LIN {X 0,Y 190.572,Z 604.003,A -85,B 0,C 180,E1 -22072.137,E2 -22072.137} C_VEL
LIN {X 0,Y 192.954,Z 597.043,A -85,B 0,C 180,E1 -22074.763,E2 -22074.763} C_VEL
LIN {X 0,Y 195.805,Z 588.854,A -85,B 0,C 180,E1 -22077.234,E2 -22077.234} C_VEL
LIN {X 0,Y 199.1,Z 578.871,A -85,B 0,C 180,E1 -22079.616,E2 -22079.616} C_VEL
LIN {X 0,Y 202.385,Z 567.586,A -85,B 0,C 180,E1 -22081.683,E2 -22081.683} C_VEL
LIN {X 0,Y 205.101,Z 556.526,A -85,B 0,C 180,E1 -22083.247,E2 -22083.247} C_VEL
LIN {X 0,Y 207.556,Z 544.251,A -85,B 0,C 180,E1 -22084.553,E2 -22084.553} C_VEL
LIN {X 0,Y 209.563,Z 531.232,A -85,B 0,C 180,E1 -22085.496,E2 -22085.496} C_VEL
LIN {X 0,Y 210.767,Z 517.939,A -85,B 0,C 180,E1 -22086.116,E2 -22086.116} C_VEL
LIN {X 0,Y 212.898,Z 471.939,A -85,B 0,C 180,E1 -22087.602,E2 -22087.602} C_VEL
LIN {X 0,Y 211.816,Z 464.418,A -85,B 0,C 180,E1 -22088.143,E2 -22088.143} C_VEL
LIN {X 0,Y 206.005,Z 450.045,A -85,B 0,C 180,E1 -22090.051,E2 -22090.051} C_VEL
LIN {X 0,Y 199.852,Z 437.156,A -85,B 0,C 180,E1 -22092.148,E2 -22092.148} C_VEL
LIN {X 0,Y 192.449,Z 423.923,A -85,B 0,C 180,E1 -22094.837,E2 -22094.837} C_VEL
LIN {X 0,Y 188.849,Z 418.24,A -85,B 0,C 180,E1 -22096.231,E2 -22096.231} C_VEL
LIN {X 0,Y 186.477,Z 414.323,A -85,B 0,C 180,E1 -22097.208,E2 -22097.208} C_VEL
LIN {X 0,Y 186.222,Z 413.566,A -85,B 0,C 180,E1 -22097.52,E2 -22097.52} C_VEL
LIN {X 0,Y 185.477,Z 410.874,A -85,B 0,C 180,E1 -22099.678,E2 -22099.678} C_VEL
LIN {X 0,Y 185.507,Z 410.87,A -85,B 0,C 180,E1 -22102.711,E2 -22102.711} C_VEL
LIN {X 0,Y 185.542,Z 410.868,A -85,B 0,C 180,E1 -22107.975,E2 -22107.975} C_VEL
LIN {X 0,Y 185.581,Z 410.869,A -85,B 0,C 180,E1 -22110.577,E2 -22110.577} C_VEL
LIN {X 0,Y 185.607,Z 410.861,A -85,B 0,C 180,E1 -22115.385,E2 -22115.385} C_VEL
LIN {X 0,Y 185.712,Z 410.845,A -85,B 0,C 180,E1 -22121.101,E2 -22121.101} C_VEL
LIN {X 0,Y 185.701,Z 410.845,A -85,B 0,C 180,E1 -22124.638,E2 -22124.638} C_VEL
LIN {X 0,Y 185.889,Z 410.823,A -85,B 0,C 180,E1 -22129.418,E2 -22129.418} C_VEL
LIN {X 0,Y 185.947,Z 410.822,A -85,B 0,C 180,E1 -22133.489,E2 -22133.489} C_VEL
LIN {X 0,Y 186.208,Z 410.789,A -85,B 0,C 180,E1 -22137.837,E2 -22137.837} C_VEL
LIN {X 0,Y 186.409,Z 410.757,A -85,B 0,C 180,E1 -22140,E2 -22140} C_VEL
LIN {X 0,Y 185.932,Z 410.824,A -85,B 0,C 180,E1 -22144.336,E2 -22144.336} C_VEL
LIN {X 0,Y 186.031,Z 410.813,A -85,B 0,C 180,E1 -22148.692,E2 -22148.692} C_VEL
LIN {X 0,Y 185.767,Z 410.841,A -85,B 0,C 180,E1 -22153.12,E2 -22153.12} C_VEL
LIN {X 0,Y 185.719,Z 410.842,A -85,B 0,C 180,E1 -22157.622,E2 -22157.622} C_VEL
LIN {X 0,Y 185.617,Z 410.856,A -85,B 0,C 180,E1 -22162.249,E2 -22162.249} C_VEL
LIN {X 0,Y 185.565,Z 410.865,A -85,B 0,C 180,E1 -22167.032,E2 -22167.032} C_VEL
LIN {X 0,Y 185.58,Z 410.864,A -85,B 0,C 180,E1 -22169.493,E2 -22169.493} C_VEL
LIN {X 0,Y 185.52,Z 410.869,A -85,B 0,C 180,E1 -22174.628,E2 -22174.628} C_VEL
LIN {X 0,Y 185.545,Z 410.866,A -85,B 0,C 180,E1 -22177.304,E2 -22177.304} C_VEL
LIN {X 0,Y 185.444,Z 410.885,A -85,B 0,C 180,E1 -22182.546,E2 -22182.546} C_VEL
LIN {X 0,Y 185.514,Z 411.362,A -85,B 0,C 180,E1 -22182.682,E2 -22182.682} C_VEL
LIN {X 0,Y 186.812,Z 414.259,A -85,B 0,C 180,E1 -22183.275,E2 -22183.275} C_VEL
LIN {X 0,Y 188.891,Z 416.481,A -85,B 0,C 180,E1 -22184.064,E2 -22184.064} C_VEL
LIN {X 0,Y 190.953,Z 419.676,A -85,B 0,C 180,E1 -22184.872,E2 -22184.872} C_VEL
LIN {X 0,Y 192.354,Z 421.693,A -85,B 0,C 180,E1 -22185.396,E2 -22185.396} C_VEL
LIN {X 0,Y 197.731,Z 429.638,A -85,B 0,C 180,E1 -22187.31,E2 -22187.31} C_VEL
LIN {X 0,Y 202.517,Z 437.59,A -85,B 0,C 180,E1 -22188.923,E2 -22188.923} C_VEL
LIN {X 0,Y 209.209,Z 451.677,A -85,B 0,C 180,E1 -22191.125,E2 -22191.125} C_VEL
LIN {X 0,Y 213.457,Z 462.043,A -85,B 0,C 180,E1 -22192.478,E2 -22192.478} C_VEL
LIN {X 0,Y 210.815,Z 514.231,A -85,B 0,C 180,E1 -22194.156,E2 -22194.156} C_VEL
LIN {X 0,Y 209.398,Z 527.372,A -85,B 0,C 180,E1 -22194.892,E2 -22194.892} C_VEL
LIN {X 0,Y 207.581,Z 539.225,A -85,B 0,C 180,E1 -22195.892,E2 -22195.892} C_VEL
LIN {X 0,Y 205.096,Z 551.651,A -85,B 0,C 180,E1 -22197.337,E2 -22197.337} C_VEL
LIN {X 0,Y 202.158,Z 563.282,A -85,B 0,C 180,E1 -22199.151,E2 -22199.151} C_VEL
LIN {X 0,Y 199.144,Z 573.728,A -85,B 0,C 180,E1 -22201.26,E2 -22201.26} C_VEL
LIN {X 0,Y 195.977,Z 583.471,A -85,B 0,C 180,E1 -22203.772,E2 -22203.772} C_VEL
LIN {X 0,Y 193.167,Z 591.508,A -85,B 0,C 180,E1 -22206.409,E2 -22206.409} C_VEL
LIN {X 0,Y 190.245,Z 598.918,A -85,B 0,C 180,E1 -22209.455,E2 -22209.455} C_VEL
LIN {X 0,Y 187.895,Z 604.861,A -85,B 0,C 180,E1 -22212.589,E2 -22212.589} C_VEL
LIN {X 0,Y 186.018,Z 609.557,A -85,B 0,C 180,E1 -22215.784,E2 -22215.784} C_VEL
LIN {X 0,Y 184.684,Z 613.147,A -85,B 0,C 180,E1 -22219.032,E2 -22219.032} C_VEL
LIN {X 0,Y 184.036,Z 615,A -85,B 0,C 180,E1 -22221.214,E2 -22221.214} C_VEL
LIN {X 0,Y 183.317,Z 617.38,A -85,B 0,C 180,E1 -22225.603,E2 -22225.603} C_VEL
LIN {X 0,Y 183.183,Z 617.988,A -85,B 0,C 180,E1 -22227.802,E2 -22227.802} C_VEL
LIN {X 0,Y 183.146,Z 618.215,A -85,B 0,C 180,E1 -22230,E2 -22230} C_VEL
LIN {X 0,Y 183.183,Z 618.02,A -85,B 0,C 180,E1 -22232.199,E2 -22232.199} C_VEL
LIN {X 0,Y 183.338,Z 617.336,A -85,B 0,C 180,E1 -22234.67,E2 -22234.67} C_VEL
LIN {X 0,Y 184.039,Z 615.106,A -85,B 0,C 180,E1 -22238.787,E2 -22238.787} C_VEL
LIN {X 0,Y 185.059,Z 612.234,A -85,B 0,C 180,E1 -22242.057,E2 -22242.057} C_VEL
LIN {X 0,Y 186.553,Z 608.338,A -85,B 0,C 180,E1 -22245.291,E2 -22245.291} C_VEL
LIN {X 0,Y 188.529,Z 603.311,A -85,B 0,C 180,E1 -22248.474,E2 -22248.474} C_VEL
LIN {X 0,Y 191.104,Z 596.975,A -85,B 0,C 180,E1 -22251.578,E2 -22251.578} C_VEL
LIN {X 0,Y 194.125,Z 589.049,A -85,B 0,C 180,E1 -22254.604,E2 -22254.604} C_VEL
LIN {X 0,Y 196.876,Z 580.943,A -85,B 0,C 180,E1 -22257.084,E2 -22257.084} C_VEL
LIN {X 0,Y 199.983,Z 571.112,A -85,B 0,C 180,E1 -22259.473,E2 -22259.473} C_VEL
LIN {X 0,Y 203.16,Z 560.003,A -85,B 0,C 180,E1 -22261.549,E2 -22261.549} C_VEL
LIN {X 0,Y 205.787,Z 549.112,A -85,B 0,C 180,E1 -22263.123,E2 -22263.123} C_VEL
LIN {X 0,Y 208.141,Z 537.07,A -85,B 0,C 180,E1 -22264.443,E2 -22264.443} C_VEL
LIN {X 0,Y 209.904,Z 524.47,A -85,B 0,C 180,E1 -22265.442,E2 -22265.442} C_VEL
LIN {X 0,Y 211.125,Z 511.734,A -85,B 0,C 180,E1 -22266.071,E2 -22266.071} C_VEL
LIN {X 0,Y 213.616,Z 462.302,A -85,B 0,C 180,E1 -22267.64,E2 -22267.64} C_VEL
LIN {X 0,Y 207.998,Z 448.85,A -85,B 0,C 180,E1 -22269.437,E2 -22269.437} C_VEL
LIN {X 0,Y 201.622,Z 435.906,A -85,B 0,C 180,E1 -22271.554,E2 -22271.554} C_VEL
LIN {X 0,Y 196.195,Z 427.311,A -85,B 0,C 180,E1 -22273.405,E2 -22273.405} C_VEL
LIN {X 0,Y 193.394,Z 423.203,A -85,B 0,C 180,E1 -22274.409,E2 -22274.409} C_VEL
LIN {X 0,Y 191.057,Z 419.751,A -85,B 0,C 180,E1 -22275.284,E2 -22275.284} C_VEL
LIN {X 0,Y 188.911,Z 416.491,A -85,B 0,C 180,E1 -22276.124,E2 -22276.124} C_VEL
LIN {X 0,Y 187.893,Z 415.362,A -85,B 0,C 180,E1 -22276.511,E2 -22276.511} C_VEL
LIN {X 0,Y 186.07,Z 412.941,A -85,B 0,C 180,E1 -22277.244,E2 -22277.244} C_VEL
LIN {X 0,Y 185.467,Z 410.881,A -85,B 0,C 180,E1 -22277.614,E2 -22277.614} C_VEL
LIN {X 0,Y 185.547,Z 410.861,A -85,B 0,C 180,E1 -22282.696,E2 -22282.696} C_VEL
LIN {X 0,Y 185.549,Z 410.873,A -85,B 0,C 180,E1 -22287.976,E2 -22287.976} C_VEL
LIN {X 0,Y 185.585,Z 410.859,A -85,B 0,C 180,E1 -22290.576,E2 -22290.576} C_VEL
LIN {X 0,Y 185.609,Z 410.852,A -85,B 0,C 180,E1 -22295.385,E2 -22295.385} C_VEL
LIN {X 0,Y 185.714,Z 410.839,A -85,B 0,C 180,E1 -22301.101,E2 -22301.101} C_VEL
LIN {X 0,Y 185.733,Z 410.846,A -85,B 0,C 180,E1 -22304.64,E2 -22304.64} C_VEL
LIN {X 0,Y 185.947,Z 410.822,A -85,B 0,C 180,E1 -22309.328,E2 -22309.328} C_VEL
LIN {X 0,Y 185.97,Z 410.805,A -85,B 0,C 180,E1 -22313.49,E2 -22313.49} C_VEL
LIN {X 0,Y 186.213,Z 410.779,A -85,B 0,C 180,E1 -22317.837,E2 -22317.837} C_VEL
LIN {X 0,Y 186.411,Z 410.751,A -85,B 0,C 180,E1 -22320,E2 -22320} C_VEL
LIN {X 0,Y 185.923,Z 410.816,A -85,B 0,C 180,E1 -22324.336,E2 -22324.336} C_VEL
LIN {X 0,Y 185.985,Z 410.817,A -85,B 0,C 180,E1 -22328.694,E2 -22328.694} C_VEL
LIN {X 0,Y 185.733,Z 410.844,A -85,B 0,C 180,E1 -22333.123,E2 -22333.123} C_VEL
LIN {X 0,Y 185.694,Z 410.843,A -85,B 0,C 180,E1 -22337.624,E2 -22337.624} C_VEL
LIN {X 0,Y 185.6,Z 410.854,A -85,B 0,C 180,E1 -22342.251,E2 -22342.251} C_VEL
LIN {X 0,Y 185.564,Z 410.871,A -85,B 0,C 180,E1 -22347.032,E2 -22347.032} C_VEL
LIN {X 0,Y 185.58,Z 410.868,A -85,B 0,C 180,E1 -22349.493,E2 -22349.493} C_VEL
LIN {X 0,Y 185.501,Z 410.874,A -85,B 0,C 180,E1 -22354.632,E2 -22354.632} C_VEL
LIN {X 0,Y 185.509,Z 410.876,A -85,B 0,C 180,E1 -22357.312,E2 -22357.312} C_VEL
LIN {X 0,Y 185.469,Z 410.881,A -85,B 0,C 180,E1 -22360.324,E2 -22360.324} C_VEL
LIN {X 0,Y 186.424,Z 414.148,A -85,B 0,C 180,E1 -22362.655,E2 -22362.655} C_VEL
LIN {X 0,Y 188.884,Z 418.272,A -85,B 0,C 180,E1 -22363.678,E2 -22363.678} C_VEL
LIN {X 0,Y 190.38,Z 420.612,A -85,B 0,C 180,E1 -22364.268,E2 -22364.268} C_VEL
LIN {X 0,Y 193.811,Z 426.389,A -85,B 0,C 180,E1 -22365.588,E2 -22365.588} C_VEL
LIN {X 0,Y 198.904,Z 435.374,A -85,B 0,C 180,E1 -22367.433,E2 -22367.433} C_VEL
LIN {X 0,Y 205.402,Z 448.544,A -85,B 0,C 180,E1 -22369.662,E2 -22369.662} C_VEL
LIN {X 0,Y 211.443,Z 463.227,A -85,B 0,C 180,E1 -22371.655,E2 -22371.655} C_VEL
LIN {X 0,Y 212.289,Z 465.956,A -85,B 0,C 180,E1 -22371.95,E2 -22371.95} C_VEL
LIN {X 0,Y 213.064,Z 474.223,A -85,B 0,C 180,E1 -22372.456,E2 -22372.456} C_VEL
LIN {X 0,Y 212.426,Z 487.121,A -85,B 0,C 180,E1 -22372.861,E2 -22372.861} C_VEL
LIN {X 0,Y 211.673,Z 492.962,A -85,B 0,C 180,E1 -22372.944,E2 -22372.944} C_VEL
LIN {X 0,Y 206.194,Z 511.984,A -85,B 0,C 180,E1 -22372.597,E2 -22372.597} C_VEL
LIN {X 0,Y 205.189,Z 517.818,A -85,B 0,C 180,E1 -22372.667,E2 -22372.667} C_VEL
LIN {X 0,Y 203.891,Z 531.383,A -85,B 0,C 180,E1 -22373.311,E2 -22373.311} C_VEL
LIN {X 0,Y 202.022,Z 543.459,A -85,B 0,C 180,E1 -22374.205,E2 -22374.205} C_VEL
LIN {X 0,Y 199.632,Z 555.008,A -85,B 0,C 180,E1 -22375.411,E2 -22375.411} C_VEL
LIN {X 0,Y 196.782,Z 566.323,A -85,B 0,C 180,E1 -22376.999,E2 -22376.999} C_VEL
LIN {X 0,Y 193.351,Z 577.834,A -85,B 0,C 180,E1 -22379.107,E2 -22379.107} C_VEL
LIN {X 0,Y 190.186,Z 587.102,A -85,B 0,C 180,E1 -22381.288,E2 -22381.288} C_VEL
LIN {X 0,Y 187.081,Z 595.557,A -85,B 0,C 180,E1 -22383.806,E2 -22383.806} C_VEL
LIN {X 0,Y 184.008,Z 603.957,A -85,B 0,C 180,E1 -22387.018,E2 -22387.018} C_VEL
LIN {X 0,Y 181.358,Z 610.477,A -85,B 0,C 180,E1 -22390.179,E2 -22390.179} C_VEL
LIN {X 0,Y 178.771,Z 616.564,A -85,B 0,C 180,E1 -22394.026,E2 -22394.026} C_VEL
LIN {X 0,Y 177.403,Z 620.528,A -85,B 0,C 180,E1 -22397.414,E2 -22397.414} C_VEL
LIN {X 0,Y 176.476,Z 623.458,A -85,B 0,C 180,E1 -22400.833,E2 -22400.833} C_VEL
LIN {X 0,Y 176.139,Z 624.853,A -85,B 0,C 180,E1 -22403.125,E2 -22403.125} C_VEL
LIN {X 0,Y 175.95,Z 626.459,A -85,B 0,C 180,E1 -22407.71,E2 -22407.71} C_VEL
LIN {X 0,Y 176.021,Z 626.672,A -85,B 0,C 180,E1 -22410,E2 -22410} C_VEL
LIN {X 0,Y 175.947,Z 626.286,A -85,B 0,C 180,E1 -22413.037,E2 -22413.037} C_VEL
LIN {X 0,Y 176.14,Z 624.824,A -85,B 0,C 180,E1 -22416.874,E2 -22416.874} C_VEL
LIN {X 0,Y 176.475,Z 623.416,A -85,B 0,C 180,E1 -22419.166,E2 -22419.166} C_VEL
LIN {X 0,Y 177.401,Z 620.467,A -85,B 0,C 180,E1 -22422.585,E2 -22422.585} C_VEL
LIN {X 0,Y 178.766,Z 616.48,A -85,B 0,C 180,E1 -22425.973,E2 -22425.973} C_VEL
LIN {X 0,Y 181.351,Z 610.36,A -85,B 0,C 180,E1 -22429.821,E2 -22429.821} C_VEL
LIN {X 0,Y 183.98,Z 603.849,A -85,B 0,C 180,E1 -22432.968,E2 -22432.968} C_VEL
LIN {X 0,Y 186.513,Z 596.873,A -85,B 0,C 180,E1 -22435.679,E2 -22435.679} C_VEL
LIN {X 0,Y 189.491,Z 588.683,A -85,B 0,C 180,E1 -22438.221,E2 -22438.221} C_VEL
LIN {X 0,Y 192.938,Z 578.7,A -85,B 0,C 180,E1 -22440.661,E2 -22440.661} C_VEL
LIN {X 0,Y 196.374,Z 567.414,A -85,B 0,C 180,E1 -22442.772,E2 -22442.772} C_VEL
LIN {X 0,Y 199.204,Z 556.353,A -85,B 0,C 180,E1 -22444.367,E2 -22444.367} C_VEL
LIN {X 0,Y 201.749,Z 544.077,A -85,B 0,C 180,E1 -22445.696,E2 -22445.696} C_VEL
LIN {X 0,Y 203.778,Z 531.507,A -85,B 0,C 180,E1 -22446.627,E2 -22446.627} C_VEL
LIN {X 0,Y 205.04,Z 518.252,A -85,B 0,C 180,E1 -22447.267,E2 -22447.267} C_VEL
LIN {X 0,Y 207.279,Z 472.993,A -85,B 0,C 180,E1 -22448.754,E2 -22448.754} C_VEL
LIN {X 0,Y 206.377,Z 466.975,A -85,B 0,C 180,E1 -22449.218,E2 -22449.218} C_VEL
LIN {X 0,Y 200.979,Z 453.477,A -85,B 0,C 180,E1 -22451.099,E2 -22451.099} C_VEL
LIN {X 0,Y 195.129,Z 441.074,A -85,B 0,C 180,E1 -22453.213,E2 -22453.213} C_VEL
LIN {X 0,Y 188.378,Z 428.76,A -85,B 0,C 180,E1 -22455.815,E2 -22455.815} C_VEL
LIN {X 0,Y 181.983,Z 418.515,A -85,B 0,C 180,E1 -22458.505,E2 -22458.505} C_VEL
LIN {X 0,Y 179.496,Z 414.781,A -85,B 0,C 180,E1 -22459.629,E2 -22459.629} C_VEL
LIN {X 0,Y 178.901,Z 413.578,A -85,B 0,C 180,E1 -22459.963,E2 -22459.963} C_VEL
LIN {X 0,Y 178.402,Z 411.755,A -85,B 0,C 180,E1 -22461.549,E2 -22461.549} C_VEL
LIN {X 0,Y 178.486,Z 411.749,A -85,B 0,C 180,E1 -22466.547,E2 -22466.547} C_VEL
LIN {X 0,Y 178.522,Z 411.746,A -85,B 0,C 180,E1 -22470.007,E2 -22470.007} C_VEL
LIN {X 0,Y 178.535,Z 411.745,A -85,B 0,C 180,E1 -22474.876,E2 -22474.876} C_VEL
LIN {X 0,Y 178.655,Z 411.723,A -85,B 0,C 180,E1 -22480.755,E2 -22480.755} C_VEL
LIN {X 0,Y 178.661,Z 411.723,A -85,B 0,C 180,E1 -22486.348,E2 -22486.348} C_VEL
LIN {X 0,Y 178.911,Z 411.69,A -85,B 0,C 180,E1 -22490.96,E2 -22490.96} C_VEL
LIN {X 0,Y 179.153,Z 411.668,A -85,B 0,C 180,E1 -22497.752,E2 -22497.752} C_VEL
LIN {X 0,Y 179.372,Z 411.633,A -85,B 0,C 180,E1 -22500,E2 -22500} C_VEL
LIN {X 0,Y 178.88,Z 411.701,A -85,B 0,C 180,E1 -22504.507,E2 -22504.507} C_VEL
LIN {X 0,Y 178.98,Z 411.69,A -85,B 0,C 180,E1 -22509.037,E2 -22509.037} C_VEL
LIN {X 0,Y 178.69,Z 411.724,A -85,B 0,C 180,E1 -22513.65,E2 -22513.65} C_VEL
LIN {X 0,Y 178.681,Z 411.723,A -85,B 0,C 180,E1 -22518.341,E2 -22518.341} C_VEL
LIN {X 0,Y 178.532,Z 411.744,A -85,B 0,C 180,E1 -22523.182,E2 -22523.182} C_VEL
LIN {X 0,Y 178.489,Z 411.753,A -85,B 0,C 180,E1 -22528.197,E2 -22528.197} C_VEL
LIN {X 0,Y 178.48,Z 411.746,A -85,B 0,C 180,E1 -22530.791,E2 -22530.791} C_VEL
LIN {X 0,Y 178.497,Z 411.743,A -85,B 0,C 180,E1 -22534.225,E2 -22534.225} C_VEL
LIN {X 0,Y 178.431,Z 411.757,A -85,B 0,C 180,E1 -22539.796,E2 -22539.796} C_VEL
LIN {X 0,Y 178.446,Z 411.752,A -85,B 0,C 180,E1 -22540.16,E2 -22540.16} C_VEL
LIN {X 0,Y 179.377,Z 414.488,A -85,B 0,C 180,E1 -22540.685,E2 -22540.685} C_VEL
LIN {X 0,Y 181.412,Z 416.708,A -85,B 0,C 180,E1 -22541.563,E2 -22541.563} C_VEL
LIN {X 0,Y 184.264,Z 420.892,A -85,B 0,C 180,E1 -22542.796,E2 -22542.796} C_VEL
LIN {X 0,Y 185.603,Z 422.698,A -85,B 0,C 180,E1 -22543.344,E2 -22543.344} C_VEL
LIN {X 0,Y 191.446,Z 431.245,A -85,B 0,C 180,E1 -22545.62,E2 -22545.62} C_VEL
LIN {X 0,Y 197.09,Z 440.277,A -85,B 0,C 180,E1 -22547.654,E2 -22547.654} C_VEL
LIN {X 0,Y 203.052,Z 452.692,A -85,B 0,C 180,E1 -22549.747,E2 -22549.747} C_VEL
LIN {X 0,Y 207.787,Z 464.054,A -85,B 0,C 180,E1 -22551.346,E2 -22551.346} C_VEL
LIN {X 0,Y 205.089,Z 514.652,A -85,B 0,C 180,E1 -22553.007,E2 -22553.007} C_VEL
LIN {X 0,Y 203.546,Z 528.236,A -85,B 0,C 180,E1 -22553.795,E2 -22553.795} C_VEL
LIN {X 0,Y 201.56,Z 540.528,A -85,B 0,C 180,E1 -22554.878,E2 -22554.878} C_VEL
LIN {X 0,Y 199.163,Z 551.823,A -85,B 0,C 180,E1 -22556.236,E2 -22556.236} C_VEL
LIN {X 0,Y 196.107,Z 563.453,A -85,B 0,C 180,E1 -22558.089,E2 -22558.089} C_VEL
LIN {X 0,Y 192.944,Z 573.898,A -85,B 0,C 180,E1 -22560.245,E2 -22560.245} C_VEL
LIN {X 0,Y 189.715,Z 583.429,A -85,B 0,C 180,E1 -22562.759,E2 -22562.759} C_VEL
LIN {X 0,Y 186.677,Z 591.678,A -85,B 0,C 180,E1 -22565.536,E2 -22565.536} C_VEL
LIN {X 0,Y 183.624,Z 599.087,A -85,B 0,C 180,E1 -22568.679,E2 -22568.679} C_VEL
LIN {X 0,Y 181.112,Z 605.03,A -85,B 0,C 180,E1 -22571.915,E2 -22571.915} C_VEL
LIN {X 0,Y 179.134,Z 609.725,A -85,B 0,C 180,E1 -22575.226,E2 -22575.226} C_VEL
LIN {X 0,Y 177.702,Z 613.315,A -85,B 0,C 180,E1 -22578.595,E2 -22578.595} C_VEL
LIN {X 0,Y 177.033,Z 615.167,A -85,B 0,C 180,E1 -22580.863,E2 -22580.863} C_VEL
LIN {X 0,Y 176.262,Z 617.547,A -85,B 0,C 180,E1 -22585.427,E2 -22585.427} C_VEL
LIN {X 0,Y 176.099,Z 618.155,A -85,B 0,C 180,E1 -22587.713,E2 -22587.713} C_VEL
LIN {X 0,Y 176.057,Z 618.382,A -85,B 0,C 180,E1 -22590,E2 -22590} C_VEL
LIN {X 0,Y 176.099,Z 618.187,A -85,B 0,C 180,E1 -22592.288,E2 -22592.288} C_VEL
LIN {X 0,Y 176.232,Z 617.6,A -85,B 0,C 180,E1 -22594.575,E2 -22594.575} C_VEL
LIN {X 0,Y 177.036,Z 615.272,A -85,B 0,C 180,E1 -22599.137,E2 -22599.137} C_VEL
LIN {X 0,Y 178.123,Z 612.4,A -85,B 0,C 180,E1 -22602.534,E2 -22602.534} C_VEL
LIN {X 0,Y 179.703,Z 608.504,A -85,B 0,C 180,E1 -22605.889,E2 -22605.889} C_VEL
LIN {X 0,Y 181.808,Z 603.476,A -85,B 0,C 180,E1 -22609.183,E2 -22609.183} C_VEL
LIN {X 0,Y 184.519,Z 597.14,A -85,B 0,C 180,E1 -22612.389,E2 -22612.389} C_VEL
LIN {X 0,Y 187.661,Z 589.215,A -85,B 0,C 180,E1 -22615.511,E2 -22615.511} C_VEL
LIN {X 0,Y 190.501,Z 581.314,A -85,B 0,C 180,E1 -22617.999,E2 -22617.999} C_VEL
LIN {X 0,Y 193.836,Z 571.276,A -85,B 0,C 180,E1 -22620.505,E2 -22620.505} C_VEL
LIN {X 0,Y 197.151,Z 560.165,A -85,B 0,C 180,E1 -22622.628,E2 -22622.628} C_VEL
LIN {X 0,Y 199.882,Z 549.273,A -85,B 0,C 180,E1 -22624.234,E2 -22624.234} C_VEL
LIN {X 0,Y 202.318,Z 537.23,A -85,B 0,C 180,E1 -22625.582,E2 -22625.582} C_VEL
LIN {X 0,Y 204.211,Z 524.37,A -85,B 0,C 180,E1 -22626.609,E2 -22626.609} C_VEL
LIN {X 0,Y 205.488,Z 511.156,A -85,B 0,C 180,E1 -22627.262,E2 -22627.262} C_VEL
LIN {X 0,Y 207.921,Z 464.197,A -85,B 0,C 180,E1 -22628.784,E2 -22628.784} C_VEL
LIN {X 0,Y 202.209,Z 450.62,A -85,B 0,C 180,E1 -22630.725,E2 -22630.725} C_VEL
LIN {X 0,Y 196.625,Z 439.377,A -85,B 0,C 180,E1 -22632.695,E2 -22632.695} C_VEL
LIN {X 0,Y 190.415,Z 429.547,A -85,B 0,C 180,E1 -22634.965,E2 -22634.965} C_VEL
LIN {X 0,Y 184.567,Z 421.113,A -85,B 0,C 180,E1 -22637.291,E2 -22637.291} C_VEL
LIN {X 0,Y 182.337,Z 418.107,A -85,B 0,C 180,E1 -22638.234,E2 -22638.234} C_VEL
LIN {X 0,Y 181.448,Z 416.707,A -85,B 0,C 180,E1 -22638.633,E2 -22638.633} C_VEL
LIN {X 0,Y 179.397,Z 414.447,A -85,B 0,C 180,E1 -22639.523,E2 -22639.523} C_VEL
LIN {X 0,Y 178.46,Z 411.725,A -85,B 0,C 180,E1 -22640.12,E2 -22640.12} C_VEL
LIN {X 0,Y 178.499,Z 411.742,A -85,B 0,C 180,E1 -22645.775,E2 -22645.775} C_VEL
LIN {X 0,Y 178.526,Z 411.738,A -85,B 0,C 180,E1 -22650.006,E2 -22650.006} C_VEL
LIN {X 0,Y 178.538,Z 411.733,A -85,B 0,C 180,E1 -22654.876,E2 -22654.876} C_VEL
LIN {X 0,Y 178.658,Z 411.717,A -85,B 0,C 180,E1 -22660.755,E2 -22660.755} C_VEL
LIN {X 0,Y 178.68,Z 411.727,A -85,B 0,C 180,E1 -22664.018,E2 -22664.018} C_VEL
LIN {X 0,Y 178.899,Z 411.7,A -85,B 0,C 180,E1 -22669.153,E2 -22669.153} C_VEL
LIN {X 0,Y 178.935,Z 411.68,A -85,B 0,C 180,E1 -22673.233,E2 -22673.233} C_VEL
LIN {X 0,Y 179.159,Z 411.658,A -85,B 0,C 180,E1 -22677.752,E2 -22677.752} C_VEL
LIN {X 0,Y 179.374,Z 411.627,A -85,B 0,C 180,E1 -22680,E2 -22680} C_VEL
LIN {X 0,Y 178.871,Z 411.692,A -85,B 0,C 180,E1 -22684.507,E2 -22684.507} C_VEL
LIN {X 0,Y 178.914,Z 411.699,A -85,B 0,C 180,E1 -22689.04,E2 -22689.04} C_VEL
LIN {X 0,Y 178.662,Z 411.727,A -85,B 0,C 180,E1 -22693.652,E2 -22693.652} C_VEL
LIN {X 0,Y 178.627,Z 411.733,A -85,B 0,C 180,E1 -22699.216,E2 -22699.216} C_VEL
LIN {X 0,Y 178.537,Z 411.746,A -85,B 0,C 180,E1 -22705.124,E2 -22705.124} C_VEL
LIN {X 0,Y 178.48,Z 411.75,A -85,B 0,C 180,E1 -22710.791,E2 -22710.791} C_VEL
LIN {X 0,Y 178.487,Z 411.749,A -85,B 0,C 180,E1 -22714.219,E2 -22714.219} C_VEL
LIN {X 0,Y 178.411,Z 411.802,A -85,B 0,C 180,E1 -22718.449,E2 -22718.449} C_VEL
LIN {X 0,Y 179.015,Z 413.784,A -85,B 0,C 180,E1 -22720.006,E2 -22720.006} C_VEL
LIN {X 0,Y 181.346,Z 417.754,A -85,B 0,C 180,E1 -22721.106,E2 -22721.106} C_VEL
LIN {X 0,Y 182.923,Z 419.849,A -85,B 0,C 180,E1 -22721.787,E2 -22721.787} C_VEL
LIN {X 0,Y 186.834,Z 426.344,A -85,B 0,C 180,E1 -22723.461,E2 -22723.461} C_VEL
LIN {X 0,Y 191.428,Z 434.096,A -85,B 0,C 180,E1 -22725.287,E2 -22725.287} C_VEL
LIN {X 0,Y 197.531,Z 445.859,A -85,B 0,C 180,E1 -22727.575,E2 -22727.575} C_VEL
LIN {X 0,Y 203.228,Z 458.646,A -85,B 0,C 180,E1 -22729.602,E2 -22729.602} C_VEL
LIN {X 0,Y 206.798,Z 467.957,A -85,B 0,C 180,E1 -22730.843,E2 -22730.843} C_VEL
LIN {X 0,Y 207.45,Z 473.974,A -85,B 0,C 180,E1 -22731.25,E2 -22731.25} C_VEL
LIN {X 0,Y 205.189,Z 517.818,A -85,B 0,C 180,E1 -22732.667,E2 -22732.667} C_VEL
LIN {X 0,Y 204.063,Z 523.622,A -85,B 0,C 180,E1 -22732.753,E2 -22732.753} C_VEL
LIN {X 0,Y 200.646,Z 532.949,A -85,B 0,C 180,E1 -22732.763,E2 -22732.763} C_VEL
LIN {X 0,Y 196.974,Z 542.149,A -85,B 0,C 180,E1 -22732.994,E2 -22732.994} C_VEL
LIN {X 0,Y 195.437,Z 547.622,A -85,B 0,C 180,E1 -22733.41,E2 -22733.41} C_VEL
LIN {X 0,Y 192.494,Z 560.045,A -85,B 0,C 180,E1 -22734.897,E2 -22734.897} C_VEL
LIN {X 0,Y 189.231,Z 571.6,A -85,B 0,C 180,E1 -22736.782,E2 -22736.782} C_VEL
LIN {X 0,Y 185.761,Z 582.006,A -85,B 0,C 180,E1 -22738.97,E2 -22738.97} C_VEL
LIN {X 0,Y 182.607,Z 590.515,A -85,B 0,C 180,E1 -22741.243,E2 -22741.243} C_VEL
LIN {X 0,Y 179.548,Z 598.369,A -85,B 0,C 180,E1 -22743.873,E2 -22743.873} C_VEL
LIN {X 0,Y 176.493,Z 606.043,A -85,B 0,C 180,E1 -22747.154,E2 -22747.154} C_VEL
LIN {X 0,Y 173.4,Z 613.122,A -85,B 0,C 180,E1 -22751.08,E2 -22751.08} C_VEL
LIN {X 0,Y 171.36,Z 617.831,A -85,B 0,C 180,E1 -22754.538,E2 -22754.538} C_VEL
LIN {X 0,Y 170.063,Z 621.434,A -85,B 0,C 180,E1 -22758.075,E2 -22758.075} C_VEL
LIN {X 0,Y 169.435,Z 623.291,A -85,B 0,C 180,E1 -22760.449,E2 -22760.449} C_VEL
LIN {X 0,Y 169.074,Z 624.686,A -85,B 0,C 180,E1 -22762.836,E2 -22762.836} C_VEL
LIN {X 0,Y 168.859,Z 626.292,A -85,B 0,C 180,E1 -22767.614,E2 -22767.614} C_VEL
LIN {X 0,Y 168.934,Z 626.505,A -85,B 0,C 180,E1 -22770,E2 -22770} C_VEL
LIN {X 0,Y 168.85,Z 626.229,A -85,B 0,C 180,E1 -22772.627,E2 -22772.627} C_VEL
LIN {X 0,Y 169.075,Z 624.656,A -85,B 0,C 180,E1 -22777.163,E2 -22777.163} C_VEL
LIN {X 0,Y 169.434,Z 623.247,A -85,B 0,C 180,E1 -22779.55,E2 -22779.55} C_VEL
LIN {X 0,Y 170.445,Z 620.299,A -85,B 0,C 180,E1 -22783.107,E2 -22783.107} C_VEL
LIN {X 0,Y 171.925,Z 616.311,A -85,B 0,C 180,E1 -22786.627,E2 -22786.627} C_VEL
LIN {X 0,Y 174.661,Z 610.191,A -85,B 0,C 180,E1 -22790.614,E2 -22790.614} C_VEL
LIN {X 0,Y 177.551,Z 603.404,A -85,B 0,C 180,E1 -22793.988,E2 -22793.988} C_VEL
LIN {X 0,Y 180.696,Z 595.212,A -85,B 0,C 180,E1 -22797.194,E2 -22797.194} C_VEL
LIN {X 0,Y 183.95,Z 586.709,A -85,B 0,C 180,E1 -22799.78,E2 -22799.78} C_VEL
LIN {X 0,Y 187.635,Z 576.207,A -85,B 0,C 180,E1 -22802.259,E2 -22802.259} C_VEL
LIN {X 0,Y 191.286,Z 564.385,A -85,B 0,C 180,E1 -22804.394,E2 -22804.394} C_VEL
LIN {X 0,Y 194.249,Z 552.463,A -85,B 0,C 180,E1 -22806.01,E2 -22806.01} C_VEL
LIN {X 0,Y 196.749,Z 540.053,A -85,B 0,C 180,E1 -22807.23,E2 -22807.23} C_VEL
LIN {X 0,Y 198.669,Z 527.329,A -85,B 0,C 180,E1 -22808.08,E2 -22808.08} C_VEL
LIN {X 0,Y 199.785,Z 512.619,A -85,B 0,C 180,E1 -22808.683,E2 -22808.683} C_VEL
LIN {X 0,Y 201.745,Z 474.092,A -85,B 0,C 180,E1 -22809.969,E2 -22809.969} C_VEL
LIN {X 0,Y 201.098,Z 469.719,A -85,B 0,C 180,E1 -22810.322,E2 -22810.322} C_VEL
LIN {X 0,Y 195.588,Z 455.883,A -85,B 0,C 180,E1 -22812.365,E2 -22812.365} C_VEL
LIN {X 0,Y 190.431,Z 444.902,A -85,B 0,C 180,E1 -22814.35,E2 -22814.35} C_VEL
LIN {X 0,Y 184.192,Z 433.392,A -85,B 0,C 180,E1 -22816.904,E2 -22816.904} C_VEL
LIN {X 0,Y 178.345,Z 423.803,A -85,B 0,C 180,E1 -22819.514,E2 -22819.514} C_VEL
LIN {X 0,Y 175.055,Z 418.775,A -85,B 0,C 180,E1 -22821.103,E2 -22821.103} C_VEL
LIN {X 0,Y 171.975,Z 414.725,A -85,B 0,C 180,E1 -22822.655,E2 -22822.655} C_VEL
LIN {X 0,Y 171.494,Z 413.324,A -85,B 0,C 180,E1 -22822.993,E2 -22822.993} C_VEL
LIN {X 0,Y 171.388,Z 412.634,A -85,B 0,C 180,E1 -22823.699,E2 -22823.699} C_VEL
LIN {X 0,Y 171.44,Z 412.624,A -85,B 0,C 180,E1 -22829.414,E2 -22829.414} C_VEL
LIN {X 0,Y 171.47,Z 412.627,A -85,B 0,C 180,E1 -22834.384,E2 -22834.384} C_VEL
LIN {X 0,Y 171.611,Z 412.6,A -85,B 0,C 180,E1 -22840.875,E2 -22840.875} C_VEL
LIN {X 0,Y 171.581,Z 412.602,A -85,B 0,C 180,E1 -22845.773,E2 -22845.773} C_VEL
LIN {X 0,Y 171.848,Z 412.568,A -85,B 0,C 180,E1 -22850.585,E2 -22850.585} C_VEL
LIN {X 0,Y 171.815,Z 412.571,A -85,B 0,C 180,E1 -22855.308,E2 -22855.308} C_VEL
LIN {X 0,Y 172.334,Z 412.509,A -85,B 0,C 180,E1 -22860,E2 -22860} C_VEL
LIN {X 0,Y 171.829,Z 412.579,A -85,B 0,C 180,E1 -22864.692,E2 -22864.692} C_VEL
LIN {X 0,Y 171.912,Z 412.571,A -85,B 0,C 180,E1 -22869.412,E2 -22869.412} C_VEL
LIN {X 0,Y 171.615,Z 412.609,A -85,B 0,C 180,E1 -22874.224,E2 -22874.224} C_VEL
LIN {X 0,Y 171.576,Z 412.614,A -85,B 0,C 180,E1 -22879.591,E2 -22879.591} C_VEL
LIN {X 0,Y 171.47,Z 412.619,A -85,B 0,C 180,E1 -22885.617,E2 -22885.617} C_VEL
LIN {X 0,Y 171.443,Z 412.622,A -85,B 0,C 180,E1 -22890.587,E2 -22890.587} C_VEL
LIN {X 0,Y 171.405,Z 412.631,A -85,B 0,C 180,E1 -22896.48,E2 -22896.48} C_VEL
LIN {X 0,Y 171.395,Z 412.628,A -85,B 0,C 180,E1 -22897.308,E2 -22897.308} C_VEL
LIN {X 0,Y 172.287,Z 415.241,A -85,B 0,C 180,E1 -22897.891,E2 -22897.891} C_VEL
LIN {X 0,Y 174.273,Z 417.501,A -85,B 0,C 180,E1 -22898.874,E2 -22898.874} C_VEL
LIN {X 0,Y 175.154,Z 418.382,A -85,B 0,C 180,E1 -22899.288,E2 -22899.288} C_VEL
LIN {X 0,Y 177.141,Z 421.538,A -85,B 0,C 180,E1 -22900.268,E2 -22900.268} C_VEL
LIN {X 0,Y 178.634,Z 423.32,A -85,B 0,C 180,E1 -22900.941,E2 -22900.941} C_VEL
LIN {X 0,Y 184.738,Z 432.117,A -85,B 0,C 180,E1 -22903.582,E2 -22903.582} C_VEL
LIN {X 0,Y 191.104,Z 441.981,A -85,B 0,C 180,E1 -22906.073,E2 -22906.073} C_VEL
LIN {X 0,Y 195.197,Z 449.766,A -85,B 0,C 180,E1 -22907.608,E2 -22907.608} C_VEL
LIN {X 0,Y 200.959,Z 463.056,A -85,B 0,C 180,E1 -22909.715,E2 -22909.715} C_VEL
LIN {X 0,Y 202.19,Z 466.041,A -85,B 0,C 180,E1 -22910.148,E2 -22910.148} C_VEL
LIN {X 0,Y 199.465,Z 515.085,A -85,B 0,C 180,E1 -22911.798,E2 -22911.798} C_VEL
LIN {X 0,Y 197.842,Z 528.541,A -85,B 0,C 180,E1 -22912.589,E2 -22912.589} C_VEL
LIN {X 0,Y 195.802,Z 540.702,A -85,B 0,C 180,E1 -22913.684,E2 -22913.684} C_VEL
LIN {X 0,Y 193.313,Z 551.995,A -85,B 0,C 180,E1 -22915.069,E2 -22915.069} C_VEL
LIN {X 0,Y 190.113,Z 563.625,A -85,B 0,C 180,E1 -22916.957,E2 -22916.957} C_VEL
LIN {X 0,Y 186.817,Z 574.069,A -85,B 0,C 180,E1 -22919.165,E2 -22919.165} C_VEL
LIN {X 0,Y 183.785,Z 582.606,A -85,B 0,C 180,E1 -22921.446,E2 -22921.446} C_VEL
LIN {X 0,Y 180.853,Z 590.462,A -85,B 0,C 180,E1 -22924.076,E2 -22924.076} C_VEL
LIN {X 0,Y 177.54,Z 598.144,A -85,B 0,C 180,E1 -22927.297,E2 -22927.297} C_VEL
LIN {X 0,Y 174.356,Z 605.2,A -85,B 0,C 180,E1 -22931.188,E2 -22931.188} C_VEL
LIN {X 0,Y 172.275,Z 609.894,A -85,B 0,C 180,E1 -22934.623,E2 -22934.623} C_VEL
LIN {X 0,Y 170.746,Z 613.483,A -85,B 0,C 180,E1 -22938.124,E2 -22938.124} C_VEL
LIN {X 0,Y 170.01,Z 615.336,A -85,B 0,C 180,E1 -22940.483,E2 -22940.483} C_VEL
LIN {X 0,Y 169.18,Z 617.715,A -85,B 0,C 180,E1 -22945.235,E2 -22945.235} C_VEL
LIN {X 0,Y 169.003,Z 618.322,A -85,B 0,C 180,E1 -22947.617,E2 -22947.617} C_VEL
LIN {X 0,Y 168.971,Z 618.549,A -85,B 0,C 180,E1 -22950,E2 -22950} C_VEL
LIN {X 0,Y 169.134,Z 617.945,A -85,B 0,C 180,E1 -22954.23,E2 -22954.23} C_VEL
LIN {X 0,Y 169.455,Z 616.799,A -85,B 0,C 180,E1 -22957.148,E2 -22957.148} C_VEL
LIN {X 0,Y 170.013,Z 615.439,A -85,B 0,C 180,E1 -22959.518,E2 -22959.518} C_VEL
LIN {X 0,Y 171.18,Z 612.567,A -85,B 0,C 180,E1 -22963.051,E2 -22963.051} C_VEL
LIN {X 0,Y 172.882,Z 608.67,A -85,B 0,C 180,E1 -22966.533,E2 -22966.533} C_VEL
LIN {X 0,Y 175.121,Z 603.642,A -85,B 0,C 180,E1 -22969.946,E2 -22969.946} C_VEL
LIN {X 0,Y 177.979,Z 597.305,A -85,B 0,C 180,E1 -22973.259,E2 -22973.259} C_VEL
LIN {X 0,Y 181.176,Z 589.59,A -85,B 0,C 180,E1 -22976.406,E2 -22976.406} C_VEL
LIN {X 0,Y 184.254,Z 581.478,A -85,B 0,C 180,E1 -22979.037,E2 -22979.037} C_VEL
LIN {X 0,Y 187.742,Z 571.44,A -85,B 0,C 180,E1 -22981.607,E2 -22981.607} C_VEL
LIN {X 0,Y 191.219,Z 560.327,A -85,B 0,C 180,E1 -22983.773,E2 -22983.773} C_VEL
LIN {X 0,Y 194.068,Z 549.434,A -85,B 0,C 180,E1 -22985.411,E2 -22985.411} C_VEL
LIN {X 0,Y 196.589,Z 537.39,A -85,B 0,C 180,E1 -22986.785,E2 -22986.785} C_VEL
LIN {X 0,Y 198.6,Z 524.333,A -85,B 0,C 180,E1 -22987.838,E2 -22987.838} C_VEL
LIN {X 0,Y 199.904,Z 511.235,A -85,B 0,C 180,E1 -22988.493,E2 -22988.493} C_VEL
LIN {X 0,Y 202.35,Z 466.21,A -85,B 0,C 180,E1 -22989.978,E2 -22989.978} C_VEL
LIN {X 0,Y 196.375,Z 452.153,A -85,B 0,C 180,E1 -22992.141,E2 -22992.141} C_VEL
LIN {X 0,Y 192.033,Z 443.516,A -85,B 0,C 180,E1 -22993.768,E2 -22993.768} C_VEL
LIN {X 0,Y 186.274,Z 434.333,A -85,B 0,C 180,E1 -22995.997,E2 -22995.997} C_VEL
LIN {X 0,Y 180.714,Z 426.272,A -85,B 0,C 180,E1 -22998.334,E2 -22998.334} C_VEL
LIN {X 0,Y 177.851,Z 422.234,A -85,B 0,C 180,E1 -22999.634,E2 -22999.634} C_VEL
LIN {X 0,Y 175.528,Z 419.078,A -85,B 0,C 180,E1 -23000.739,E2 -23000.739} C_VEL
LIN {X 0,Y 174.791,Z 417.806,A -85,B 0,C 180,E1 -23001.118,E2 -23001.118} C_VEL
LIN {X 0,Y 172.684,Z 415.846,A -85,B 0,C 180,E1 -23002.129,E2 -23002.129} C_VEL
LIN {X 0,Y 171.512,Z 413.257,A -85,B 0,C 180,E1 -23002.814,E2 -23002.814} C_VEL
LIN {X 0,Y 171.417,Z 412.621,A -85,B 0,C 180,E1 -23002.974,E2 -23002.974} C_VEL
LIN {X 0,Y 171.423,Z 412.632,A -85,B 0,C 180,E1 -23007.793,E2 -23007.793} C_VEL
LIN {X 0,Y 171.453,Z 412.618,A -85,B 0,C 180,E1 -23010.535,E2 -23010.535} C_VEL
LIN {X 0,Y 171.47,Z 412.614,A -85,B 0,C 180,E1 -23015.803,E2 -23015.803} C_VEL
LIN {X 0,Y 171.614,Z 412.594,A -85,B 0,C 180,E1 -23020.875,E2 -23020.875} C_VEL
LIN {X 0,Y 171.617,Z 412.594,A -85,B 0,C 180,E1 -23025.776,E2 -23025.776} C_VEL
LIN {X 0,Y 171.912,Z 412.568,A -85,B 0,C 180,E1 -23030.588,E2 -23030.588} C_VEL
LIN {X 0,Y 171.83,Z 412.58,A -85,B 0,C 180,E1 -23035.308,E2 -23035.308} C_VEL
LIN {X 0,Y 172.337,Z 412.503,A -85,B 0,C 180,E1 -23040,E2 -23040} C_VEL
LIN {X 0,Y 171.818,Z 412.569,A -85,B 0,C 180,E1 -23044.692,E2 -23044.692} C_VEL
LIN {X 0,Y 171.851,Z 412.576,A -85,B 0,C 180,E1 -23049.415,E2 -23049.415} C_VEL
LIN {X 0,Y 171.58,Z 412.612,A -85,B 0,C 180,E1 -23054.227,E2 -23054.227} C_VEL
LIN {X 0,Y 171.548,Z 412.616,A -85,B 0,C 180,E1 -23059.562,E2 -23059.562} C_VEL
LIN {X 0,Y 171.472,Z 412.624,A -85,B 0,C 180,E1 -23065.616,E2 -23065.616} C_VEL
LIN {X 0,Y 171.443,Z 412.626,A -85,B 0,C 180,E1 -23070.585,E2 -23070.585} C_VEL
LIN {X 0,Y 171.392,Z 412.653,A -85,B 0,C 180,E1 -23076.3,E2 -23076.3} C_VEL
LIN {X 0,Y 171.515,Z 413.375,A -85,B 0,C 180,E1 -23076.91,E2 -23076.91} C_VEL
LIN {X 0,Y 172.608,Z 415.834,A -85,B 0,C 180,E1 -23077.552,E2 -23077.552} C_VEL
LIN {X 0,Y 175.787,Z 419.77,A -85,B 0,C 180,E1 -23079.123,E2 -23079.123} C_VEL
LIN {X 0,Y 178.766,Z 424.282,A -85,B 0,C 180,E1 -23080.549,E2 -23080.549} C_VEL
LIN {X 0,Y 185.138,Z 434.96,A -85,B 0,C 180,E1 -23083.385,E2 -23083.385} C_VEL
LIN {X 0,Y 191.783,Z 447.549,A -85,B 0,C 180,E1 -23086.079,E2 -23086.079} C_VEL
LIN {X 0,Y 197.917,Z 461.266,A -85,B 0,C 180,E1 -23088.411,E2 -23088.411} C_VEL
LIN {X 0,Y 201.492,Z 470.772,A -85,B 0,C 180,E1 -23089.738,E2 -23089.738} C_VEL
LIN {X 0,Y 201.873,Z 475.713,A -85,B 0,C 180,E1 -23090.054,E2 -23090.054} C_VEL
LIN {X 0,Y 199.208,Z 522.117,A -85,B 0,C 180,E1 -23091.591,E2 -23091.591} C_VEL
LIN {X 0,Y 197.564,Z 535.751,A -85,B 0,C 180,E1 -23092.383,E2 -23092.383} C_VEL
LIN {X 0,Y 195.437,Z 547.622,A -85,B 0,C 180,E1 -23093.41,E2 -23093.41} C_VEL
LIN {X 0,Y 193.735,Z 553.066,A -85,B 0,C 180,E1 -23093.877,E2 -23093.877} C_VEL
LIN {X 0,Y 189.232,Z 561.667,A -85,B 0,C 180,E1 -23094.507,E2 -23094.507} C_VEL
LIN {X 0,Y 184.42,Z 569.864,A -85,B 0,C 180,E1 -23095.369,E2 -23095.369} C_VEL
LIN {X 0,Y 182.262,Z 574.671,A -85,B 0,C 180,E1 -23096.201,E2 -23096.201} C_VEL
LIN {X 0,Y 178.608,Z 584.831,A -85,B 0,C 180,E1 -23098.575,E2 -23098.575} C_VEL
LIN {X 0,Y 175.05,Z 593.65,A -85,B 0,C 180,E1 -23101.197,E2 -23101.197} C_VEL
LIN {X 0,Y 171.86,Z 601.339,A -85,B 0,C 180,E1 -23104.114,E2 -23104.114} C_VEL
LIN {X 0,Y 168.89,Z 608.11,A -85,B 0,C 180,E1 -23107.361,E2 -23107.361} C_VEL
LIN {X 0,Y 166.687,Z 612.956,A -85,B 0,C 180,E1 -23110.287,E2 -23110.287} C_VEL
LIN {X 0,Y 164.493,Z 617.664,A -85,B 0,C 180,E1 -23113.876,E2 -23113.876} C_VEL
LIN {X 0,Y 163.107,Z 621.267,A -85,B 0,C 180,E1 -23117.558,E2 -23117.558} C_VEL
LIN {X 0,Y 162.416,Z 623.124,A -85,B 0,C 180,E1 -23120.032,E2 -23120.032} C_VEL
LIN {X 0,Y 162.001,Z 624.518,A -85,B 0,C 180,E1 -23122.521,E2 -23122.521} C_VEL
LIN {X 0,Y 161.76,Z 626.125,A -85,B 0,C 180,E1 -23127.509,E2 -23127.509} C_VEL
LIN {X 0,Y 161.833,Z 626.338,A -85,B 0,C 180,E1 -23130,E2 -23130} C_VEL
LIN {X 0,Y 161.76,Z 626.111,A -85,B 0,C 180,E1 -23132.49,E2 -23132.49} C_VEL
LIN {X 0,Y 161.792,Z 625.493,A -85,B 0,C 180,E1 -23134.984,E2 -23134.984} C_VEL
LIN {X 0,Y 162.002,Z 624.488,A -85,B 0,C 180,E1 -23137.478,E2 -23137.478} C_VEL
LIN {X 0,Y 162.416,Z 623.079,A -85,B 0,C 180,E1 -23139.967,E2 -23139.967} C_VEL
LIN {X 0,Y 163.496,Z 620.13,A -85,B 0,C 180,E1 -23143.675,E2 -23143.675} C_VEL
LIN {X 0,Y 165.116,Z 616.142,A -85,B 0,C 180,E1 -23147.334,E2 -23147.334} C_VEL
LIN {X 0,Y 167.982,Z 610.021,A -85,B 0,C 180,E1 -23151.474,E2 -23151.474} C_VEL
LIN {X 0,Y 171.374,Z 602.439,A -85,B 0,C 180,E1 -23155.327,E2 -23155.327} C_VEL
LIN {X 0,Y 174.387,Z 595.042,A -85,B 0,C 180,E1 -23158.264,E2 -23158.264} C_VEL
LIN {X 0,Y 177.818,Z 586.539,A -85,B 0,C 180,E1 -23160.917,E2 -23160.917} C_VEL
LIN {X 0,Y 181.653,Z 576.036,A -85,B 0,C 180,E1 -23163.457,E2 -23163.457} C_VEL
LIN {X 0,Y 185.018,Z 565.643,A -85,B 0,C 180,E1 -23165.4,E2 -23165.4} C_VEL
LIN {X 0,Y 188.115,Z 554.237,A -85,B 0,C 180,E1 -23167.044,E2 -23167.044} C_VEL
LIN {X 0,Y 190.674,Z 542.481,A -85,B 0,C 180,E1 -23168.293,E2 -23168.293} C_VEL
LIN {X 0,Y 192.847,Z 529.099,A -85,B 0,C 180,E1 -23169.27,E2 -23169.27} C_VEL
LIN {X 0,Y 194.064,Z 516.375,A -85,B 0,C 180,E1 -23169.86,E2 -23169.86} C_VEL
LIN {X 0,Y 196.304,Z 475.216,A -85,B 0,C 180,E1 -23171.251,E2 -23171.251} C_VEL
LIN {X 0,Y 195.736,Z 472.036,A -85,B 0,C 180,E1 -23171.548,E2 -23171.548} C_VEL
LIN {X 0,Y 190.722,Z 459.288,A -85,B 0,C 180,E1 -23173.531,E2 -23173.531} C_VEL
LIN {X 0,Y 185.093,Z 447.219,A -85,B 0,C 180,E1 -23175.851,E2 -23175.851} C_VEL
LIN {X 0,Y 179.236,Z 436.536,A -85,B 0,C 180,E1 -23178.427,E2 -23178.427} C_VEL
LIN {X 0,Y 174.515,Z 428.682,A -85,B 0,C 180,E1 -23180.69,E2 -23180.69} C_VEL
LIN {X 0,Y 171.476,Z 423.995,A -85,B 0,C 180,E1 -23182.25,E2 -23182.25} C_VEL
LIN {X 0,Y 168.56,Z 419.915,A -85,B 0,C 180,E1 -23183.826,E2 -23183.826} C_VEL
LIN {X 0,Y 168.015,Z 418.874,A -85,B 0,C 180,E1 -23184.153,E2 -23184.153} C_VEL
LIN {X 0,Y 165.593,Z 416.743,A -85,B 0,C 180,E1 -23185.481,E2 -23185.481} C_VEL
LIN {X 0,Y 164.45,Z 414.257,A -85,B 0,C 180,E1 -23186.25,E2 -23186.25} C_VEL
LIN {X 0,Y 164.32,Z 413.511,A -85,B 0,C 180,E1 -23186.395,E2 -23186.395} C_VEL
LIN {X 0,Y 164.389,Z 413.501,A -85,B 0,C 180,E1 -23189.134,E2 -23189.134} C_VEL
LIN {X 0,Y 164.419,Z 413.504,A -85,B 0,C 180,E1 -23194.694,E2 -23194.694} C_VEL
LIN {X 0,Y 164.521,Z 413.484,A -85,B 0,C 180,E1 -23200.017,E2 -23200.017} C_VEL
LIN {X 0,Y 164.532,Z 413.479,A -85,B 0,C 180,E1 -23205.15,E2 -23205.15} C_VEL
LIN {X 0,Y 164.768,Z 413.45,A -85,B 0,C 180,E1 -23210.176,E2 -23210.176} C_VEL
LIN {X 0,Y 164.831,Z 413.454,A -85,B 0,C 180,E1 -23212.651,E2 -23212.651} C_VEL
LIN {X 0,Y 165.049,Z 413.424,A -85,B 0,C 180,E1 -23217.56,E2 -23217.56} C_VEL
LIN {X 0,Y 165.297,Z 413.385,A -85,B 0,C 180,E1 -23220,E2 -23220} C_VEL
LIN {X 0,Y 164.779,Z 413.455,A -85,B 0,C 180,E1 -23224.894,E2 -23224.894} C_VEL
LIN {X 0,Y 164.864,Z 413.439,A -85,B 0,C 180,E1 -23227.348,E2 -23227.348} C_VEL
LIN {X 0,Y 164.781,Z 413.449,A -85,B 0,C 180,E1 -23231.198,E2 -23231.198} C_VEL
LIN {X 0,Y 164.527,Z 413.48,A -85,B 0,C 180,E1 -23237.399,E2 -23237.399} C_VEL
LIN {X 0,Y 164.521,Z 413.49,A -85,B 0,C 180,E1 -23239.983,E2 -23239.983} C_VEL
LIN {X 0,Y 164.395,Z 413.499,A -85,B 0,C 180,E1 -23246.135,E2 -23246.135} C_VEL
LIN {X 0,Y 164.377,Z 413.504,A -85,B 0,C 180,E1 -23251.229,E2 -23251.229} C_VEL
LIN {X 0,Y 164.356,Z 413.667,A -85,B 0,C 180,E1 -23254.033,E2 -23254.033} C_VEL
LIN {X 0,Y 165.165,Z 415.983,A -85,B 0,C 180,E1 -23254.624,E2 -23254.624} C_VEL
LIN {X 0,Y 167.104,Z 418.287,A -85,B 0,C 180,E1 -23255.749,E2 -23255.749} C_VEL
LIN {X 0,Y 168.241,Z 419.123,A -85,B 0,C 180,E1 -23256.346,E2 -23256.346} C_VEL
LIN {X 0,Y 170.277,Z 422.467,A -85,B 0,C 180,E1 -23257.502,E2 -23257.502} C_VEL
LIN {X 0,Y 172.115,Z 424.5,A -85,B 0,C 180,E1 -23258.432,E2 -23258.432} C_VEL
LIN {X 0,Y 174.795,Z 428.174,A -85,B 0,C 180,E1 -23259.766,E2 -23259.766} C_VEL
LIN {X 0,Y 181.132,Z 437.498,A -85,B 0,C 180,E1 -23262.672,E2 -23262.672} C_VEL
LIN {X 0,Y 187.279,Z 447.274,A -85,B 0,C 180,E1 -23265.208,E2 -23265.208} C_VEL
LIN {X 0,Y 191.45,Z 455.68,A -85,B 0,C 180,E1 -23266.869,E2 -23266.869} C_VEL
LIN {X 0,Y 196.725,Z 468.298,A -85,B 0,C 180,E1 -23268.904,E2 -23268.904} C_VEL
LIN {X 0,Y 193.976,Z 514.934,A -85,B 0,C 180,E1 -23270.486,E2 -23270.486} C_VEL
LIN {X 0,Y 192.32,Z 528.386,A -85,B 0,C 180,E1 -23271.284,E2 -23271.284} C_VEL
LIN {X 0,Y 190.14,Z 540.876,A -85,B 0,C 180,E1 -23272.42,E2 -23272.42} C_VEL
LIN {X 0,Y 187.536,Z 552.168,A -85,B 0,C 180,E1 -23273.826,E2 -23273.826} C_VEL
LIN {X 0,Y 184.214,Z 563.796,A -85,B 0,C 180,E1 -23275.755,E2 -23275.755} C_VEL
LIN {X 0,Y 180.77,Z 574.239,A -85,B 0,C 180,E1 -23278.014,E2 -23278.014} C_VEL
LIN {X 0,Y 177.192,Z 583.814,A -85,B 0,C 180,E1 -23280.672,E2 -23280.672} C_VEL
LIN {X 0,Y 173.845,Z 592.017,A -85,B 0,C 180,E1 -23283.596,E2 -23283.596} C_VEL
LIN {X 0,Y 170.496,Z 599.424,A -85,B 0,C 180,E1 -23286.946,E2 -23286.946} C_VEL
LIN {X 0,Y 167.634,Z 605.369,A -85,B 0,C 180,E1 -23290.404,E2 -23290.404} C_VEL
LIN {X 0,Y 165.444,Z 610.062,A -85,B 0,C 180,E1 -23293.972,E2 -23293.972} C_VEL
LIN {X 0,Y 163.787,Z 613.651,A -85,B 0,C 180,E1 -23297.611,E2 -23297.611} C_VEL
LIN {X 0,Y 163.002,Z 615.504,A -85,B 0,C 180,E1 -23300.069,E2 -23300.069} C_VEL
LIN {X 0,Y 162.109,Z 617.882,A -85,B 0,C 180,E1 -23305.026,E2 -23305.026} C_VEL
LIN {X 0,Y 161.926,Z 618.489,A -85,B 0,C 180,E1 -23307.513,E2 -23307.513} C_VEL
LIN {X 0,Y 161.887,Z 618.716,A -85,B 0,C 180,E1 -23310,E2 -23310} C_VEL
LIN {X 0,Y 162.029,Z 618.242,A -85,B 0,C 180,E1 -23313.943,E2 -23313.943} C_VEL
LIN {X 0,Y 162.407,Z 616.966,A -85,B 0,C 180,E1 -23317.46,E2 -23317.46} C_VEL
LIN {X 0,Y 163.005,Z 615.606,A -85,B 0,C 180,E1 -23319.931,E2 -23319.931} C_VEL
LIN {X 0,Y 164.261,Z 612.733,A -85,B 0,C 180,E1 -23323.611,E2 -23323.611} C_VEL
LIN {X 0,Y 166.091,Z 608.836,A -85,B 0,C 180,E1 -23327.23,E2 -23327.23} C_VEL
LIN {X 0,Y 168.471,Z 603.807,A -85,B 0,C 180,E1 -23330.769,E2 -23330.769} C_VEL
LIN {X 0,Y 171.488,Z 597.47,A -85,B 0,C 180,E1 -23334.194,E2 -23334.194} C_VEL
LIN {X 0,Y 174.713,Z 590.043,A -85,B 0,C 180,E1 -23337.337,E2 -23337.337} C_VEL
LIN {X 0,Y 178.148,Z 581.467,A -85,B 0,C 180,E1 -23340.198,E2 -23340.198} C_VEL
LIN {X 0,Y 181.739,Z 571.603,A -85,B 0,C 180,E1 -23342.779,E2 -23342.779} C_VEL
LIN {X 0,Y 185.362,Z 560.49,A -85,B 0,C 180,E1 -23344.993,E2 -23344.993} C_VEL
LIN {X 0,Y 188.34,Z 549.595,A -85,B 0,C 180,E1 -23346.66,E2 -23346.66} C_VEL
LIN {X 0,Y 190.96,Z 537.549,A -85,B 0,C 180,E1 -23348.059,E2 -23348.059} C_VEL
LIN {X 0,Y 192.975,Z 524.983,A -85,B 0,C 180,E1 -23349.101,E2 -23349.101} C_VEL
LIN {X 0,Y 194.366,Z 511.95,A -85,B 0,C 180,E1 -23349.771,E2 -23349.771} C_VEL
LIN {X 0,Y 196.879,Z 468.419,A -85,B 0,C 180,E1 -23351.228,E2 -23351.228} C_VEL
LIN {X 0,Y 191.083,Z 454.666,A -85,B 0,C 180,E1 -23353.473,E2 -23353.473} C_VEL
LIN {X 0,Y 187.075,Z 446.837,A -85,B 0,C 180,E1 -23355.071,E2 -23355.071} C_VEL
LIN {X 0,Y 180.137,Z 435.872,A -85,B 0,C 180,E1 -23357.977,E2 -23357.977} C_VEL
LIN {X 0,Y 174.363,Z 427.65,A -85,B 0,C 180,E1 -23360.661,E2 -23360.661} C_VEL
LIN {X 0,Y 171.316,Z 423.471,A -85,B 0,C 180,E1 -23362.208,E2 -23362.208} C_VEL
LIN {X 0,Y 168.847,Z 420.346,A -85,B 0,C 180,E1 -23363.527,E2 -23363.527} C_VEL
LIN {X 0,Y 168.085,Z 418.893,A -85,B 0,C 180,E1 -23363.986,E2 -23363.986} C_VEL
LIN {X 0,Y 165.712,Z 416.845,A -85,B 0,C 180,E1 -23365.289,E2 -23365.289} C_VEL
LIN {X 0,Y 164.548,Z 414.488,A -85,B 0,C 180,E1 -23366.063,E2 -23366.063} C_VEL
LIN {X 0,Y 164.347,Z 413.504,A -85,B 0,C 180,E1 -23366.313,E2 -23366.313} C_VEL
LIN {X 0,Y 164.394,Z 413.502,A -85,B 0,C 180,E1 -23369.135,E2 -23369.135} C_VEL
LIN {X 0,Y 164.422,Z 413.492,A -85,B 0,C 180,E1 -23374.695,E2 -23374.695} C_VEL
LIN {X 0,Y 164.524,Z 413.478,A -85,B 0,C 180,E1 -23380.017,E2 -23380.017} C_VEL
LIN {X 0,Y 164.563,Z 413.476,A -85,B 0,C 180,E1 -23385.153,E2 -23385.153} C_VEL
LIN {X 0,Y 164.855,Z 413.449,A -85,B 0,C 180,E1 -23390.181,E2 -23390.181} C_VEL
LIN {X 0,Y 164.78,Z 413.458,A -85,B 0,C 180,E1 -23395.107,E2 -23395.107} C_VEL
LIN {X 0,Y 165.299,Z 413.379,A -85,B 0,C 180,E1 -23400,E2 -23400} C_VEL
LIN {X 0,Y 164.767,Z 413.445,A -85,B 0,C 180,E1 -23404.894,E2 -23404.894} C_VEL
LIN {X 0,Y 164.834,Z 413.446,A -85,B 0,C 180,E1 -23407.349,E2 -23407.349} C_VEL
LIN {X 0,Y 164.706,Z 413.454,A -85,B 0,C 180,E1 -23411.061,E2 -23411.061} C_VEL
LIN {X 0,Y 164.487,Z 413.482,A -85,B 0,C 180,E1 -23417.403,E2 -23417.403} C_VEL
LIN {X 0,Y 164.477,Z 413.498,A -85,B 0,C 180,E1 -23419.989,E2 -23419.989} C_VEL
LIN {X 0,Y 164.396,Z 413.505,A -85,B 0,C 180,E1 -23426.133,E2 -23426.133} C_VEL
LIN {X 0,Y 164.381,Z 413.505,A -85,B 0,C 180,E1 -23432.374,E2 -23432.374} C_VEL
LIN {X 0,Y 164.342,Z 413.512,A -85,B 0,C 180,E1 -23433.425,E2 -23433.425} C_VEL
LIN {X 0,Y 165.18,Z 416.079,A -85,B 0,C 180,E1 -23434.098,E2 -23434.098} C_VEL
LIN {X 0,Y 167.164,Z 418.335,A -85,B 0,C 180,E1 -23435.249,E2 -23435.249} C_VEL
LIN {X 0,Y 168.31,Z 419.347,A -85,B 0,C 180,E1 -23435.866,E2 -23435.866} C_VEL
LIN {X 0,Y 170.349,Z 422.56,A -85,B 0,C 180,E1 -23437.02,E2 -23437.02} C_VEL
LIN {X 0,Y 172.509,Z 425.445,A -85,B 0,C 180,E1 -23438.146,E2 -23438.146} C_VEL
LIN {X 0,Y 176.348,Z 431.611,A -85,B 0,C 180,E1 -23440.082,E2 -23440.082} C_VEL
LIN {X 0,Y 181.387,Z 440.157,A -85,B 0,C 180,E1 -23442.421,E2 -23442.421} C_VEL
LIN {X 0,Y 187.515,Z 452.109,A -85,B 0,C 180,E1 -23445.058,E2 -23445.058} C_VEL
LIN {X 0,Y 193.309,Z 465.448,A -85,B 0,C 180,E1 -23447.4,E2 -23447.4} C_VEL
LIN {X 0,Y 196.265,Z 473.417,A -85,B 0,C 180,E1 -23448.566,E2 -23448.566} C_VEL
LIN {X 0,Y 196.342,Z 478.217,A -85,B 0,C 180,E1 -23448.814,E2 -23448.814} C_VEL
LIN {X 0,Y 193.658,Z 522.385,A -85,B 0,C 180,E1 -23450.308,E2 -23450.308} C_VEL
LIN {X 0,Y 191.961,Z 535.801,A -85,B 0,C 180,E1 -23451.106,E2 -23451.106} C_VEL
LIN {X 0,Y 189.508,Z 548.806,A -85,B 0,C 180,E1 -23452.271,E2 -23452.271} C_VEL
LIN {X 0,Y 186.316,Z 561.466,A -85,B 0,C 180,E1 -23453.886,E2 -23453.886} C_VEL
LIN {X 0,Y 182.921,Z 572.73,A -85,B 0,C 180,E1 -23455.811,E2 -23455.811} C_VEL
LIN {X 0,Y 182.262,Z 574.671,A -85,B 0,C 180,E1 -23456.201,E2 -23456.201} C_VEL
LIN {X 0,Y 180.034,Z 579.419,A -85,B 0,C 180,E1 -23457.118,E2 -23457.118} C_VEL
LIN {X 0,Y 174.751,Z 586.725,A -85,B 0,C 180,E1 -23458.49,E2 -23458.49} C_VEL
LIN {X 0,Y 169.429,Z 593.431,A -85,B 0,C 180,E1 -23460.116,E2 -23460.116} C_VEL
LIN {X 0,Y 167.185,Z 597.247,A -85,B 0,C 180,E1 -23461.412,E2 -23461.412} C_VEL
LIN {X 0,Y 164.024,Z 604.558,A -85,B 0,C 180,E1 -23464.629,E2 -23464.629} C_VEL
LIN {X 0,Y 160.937,Z 610.971,A -85,B 0,C 180,E1 -23468.21,E2 -23468.21} C_VEL
LIN {X 0,Y 158.344,Z 616.064,A -85,B 0,C 180,E1 -23471.898,E2 -23471.898} C_VEL
LIN {X 0,Y 156.572,Z 620.027,A -85,B 0,C 180,E1 -23475.707,E2 -23475.707} C_VEL
LIN {X 0,Y 155.419,Z 622.957,A -85,B 0,C 180,E1 -23479.578,E2 -23479.578} C_VEL
LIN {X 0,Y 154.952,Z 624.351,A -85,B 0,C 180,E1 -23482.179,E2 -23482.179} C_VEL
LIN {X 0,Y 154.665,Z 625.958,A -85,B 0,C 180,E1 -23487.395,E2 -23487.395} C_VEL
LIN {X 0,Y 154.745,Z 626.171,A -85,B 0,C 180,E1 -23490,E2 -23490} C_VEL
LIN {X 0,Y 154.665,Z 625.943,A -85,B 0,C 180,E1 -23492.604,E2 -23492.604} C_VEL
LIN {X 0,Y 154.712,Z 625.326,A -85,B 0,C 180,E1 -23495.212,E2 -23495.212} C_VEL
LIN {X 0,Y 154.952,Z 624.32,A -85,B 0,C 180,E1 -23497.82,E2 -23497.82} C_VEL
LIN {X 0,Y 155.418,Z 622.911,A -85,B 0,C 180,E1 -23500.421,E2 -23500.421} C_VEL
LIN {X 0,Y 156.57,Z 619.961,A -85,B 0,C 180,E1 -23504.293,E2 -23504.293} C_VEL
LIN {X 0,Y 158.339,Z 615.974,A -85,B 0,C 180,E1 -23508.101,E2 -23508.101} C_VEL
LIN {X 0,Y 161.336,Z 609.85,A -85,B 0,C 180,E1 -23512.405,E2 -23512.405} C_VEL
LIN {X 0,Y 164.686,Z 602.846,A -85,B 0,C 180,E1 -23516.115,E2 -23516.115} C_VEL
LIN {X 0,Y 168.151,Z 594.872,A -85,B 0,C 180,E1 -23519.413,E2 -23519.413} C_VEL
LIN {X 0,Y 171.764,Z 586.369,A -85,B 0,C 180,E1 -23522.135,E2 -23522.135} C_VEL
LIN {X 0,Y 175.768,Z 575.865,A -85,B 0,C 180,E1 -23524.734,E2 -23524.734} C_VEL
LIN {X 0,Y 179.286,Z 565.472,A -85,B 0,C 180,E1 -23526.712,E2 -23526.712} C_VEL
LIN {X 0,Y 182.497,Z 554.065,A -85,B 0,C 180,E1 -23528.387,E2 -23528.387} C_VEL
LIN {X 0,Y 185.152,Z 542.305,A -85,B 0,C 180,E1 -23529.655,E2 -23529.655} C_VEL
LIN {X 0,Y 187.405,Z 529.024,A -85,B 0,C 180,E1 -23530.634,E2 -23530.634} C_VEL
LIN {X 0,Y 188.676,Z 516.19,A -85,B 0,C 180,E1 -23531.24,E2 -23531.24} C_VEL
LIN {X 0,Y 190.966,Z 476.353,A -85,B 0,C 180,E1 -23532.604,E2 -23532.604} C_VEL
LIN {X 0,Y 189.272,Z 471.128,A -85,B 0,C 180,E1 -23533.34,E2 -23533.34} C_VEL
LIN {X 0,Y 183.65,Z 457.496,A -85,B 0,C 180,E1 -23535.749,E2 -23535.749} C_VEL
LIN {X 0,Y 178.228,Z 446.55,A -85,B 0,C 180,E1 -23538.197,E2 -23538.197} C_VEL
LIN {X 0,Y 172.664,Z 436.683,A -85,B 0,C 180,E1 -23540.923,E2 -23540.923} C_VEL
LIN {X 0,Y 168.263,Z 429.549,A -85,B 0,C 180,E1 -23543.287,E2 -23543.287} C_VEL
LIN {X 0,Y 165.303,Z 425.242,A -85,B 0,C 180,E1 -23544.993,E2 -23544.993} C_VEL
LIN {X 0,Y 162.326,Z 421.916,A -85,B 0,C 180,E1 -23546.773,E2 -23546.773} C_VEL
LIN {X 0,Y 161.22,Z 419.868,A -85,B 0,C 180,E1 -23547.538,E2 -23547.538} C_VEL
LIN {X 0,Y 158.779,Z 417.853,A -85,B 0,C 180,E1 -23549.113,E2 -23549.113} C_VEL
LIN {X 0,Y 157.551,Z 415.591,A -85,B 0,C 180,E1 -23550.063,E2 -23550.063} C_VEL
LIN {X 0,Y 157.299,Z 414.391,A -85,B 0,C 180,E1 -23550.379,E2 -23550.379} C_VEL
LIN {X 0,Y 157.322,Z 414.384,A -85,B 0,C 180,E1 -23553.466,E2 -23553.466} C_VEL
LIN {X 0,Y 157.447,Z 414.366,A -85,B 0,C 180,E1 -23559.616,E2 -23559.616} C_VEL
LIN {X 0,Y 157.465,Z 414.361,A -85,B 0,C 180,E1 -23564.467,E2 -23564.467} C_VEL
LIN {X 0,Y 157.69,Z 414.332,A -85,B 0,C 180,E1 -23569.731,E2 -23569.731} C_VEL
LIN {X 0,Y 157.768,Z 414.331,A -85,B 0,C 180,E1 -23572.32,E2 -23572.32} C_VEL
LIN {X 0,Y 158.259,Z 414.261,A -85,B 0,C 180,E1 -23580,E2 -23580} C_VEL
LIN {X 0,Y 157.826,Z 414.317,A -85,B 0,C 180,E1 -23587.677,E2 -23587.677} C_VEL
LIN {X 0,Y 157.707,Z 414.329,A -85,B 0,C 180,E1 -23591.363,E2 -23591.363} C_VEL
LIN {X 0,Y 157.489,Z 414.362,A -85,B 0,C 180,E1 -23595.531,E2 -23595.531} C_VEL
LIN {X 0,Y 157.416,Z 414.369,A -85,B 0,C 180,E1 -23600.927,E2 -23600.927} C_VEL
LIN {X 0,Y 157.316,Z 414.381,A -85,B 0,C 180,E1 -23606.686,E2 -23606.686} C_VEL
LIN {X 0,Y 157.327,Z 414.522,A -85,B 0,C 180,E1 -23610.077,E2 -23610.077} C_VEL
LIN {X 0,Y 158.277,Z 417.085,A -85,B 0,C 180,E1 -23610.894,E2 -23610.894} C_VEL
LIN {X 0,Y 160.111,Z 419.219,A -85,B 0,C 180,E1 -23612.159,E2 -23612.159} C_VEL
LIN {X 0,Y 161.53,Z 420.255,A -85,B 0,C 180,E1 -23613.04,E2 -23613.04} C_VEL
LIN {X 0,Y 163.435,Z 423.413,A -85,B 0,C 180,E1 -23614.304,E2 -23614.304} C_VEL
LIN {X 0,Y 165.494,Z 425.527,A -85,B 0,C 180,E1 -23615.498,E2 -23615.498} C_VEL
LIN {X 0,Y 168.16,Z 429.235,A -85,B 0,C 180,E1 -23617.02,E2 -23617.02} C_VEL
LIN {X 0,Y 172.465,Z 435.347,A -85,B 0,C 180,E1 -23619.286,E2 -23619.286} C_VEL
LIN {X 0,Y 177.325,Z 442.477,A -85,B 0,C 180,E1 -23621.61,E2 -23621.61} C_VEL
LIN {X 0,Y 183.323,Z 452.314,A -85,B 0,C 180,E1 -23624.238,E2 -23624.238} C_VEL
LIN {X 0,Y 187.081,Z 460.062,A -85,B 0,C 180,E1 -23625.824,E2 -23625.824} C_VEL
LIN {X 0,Y 191.295,Z 470.403,A -85,B 0,C 180,E1 -23627.565,E2 -23627.565} C_VEL
LIN {X 0,Y 188.575,Z 515.021,A -85,B 0,C 180,E1 -23629.112,E2 -23629.112} C_VEL
LIN {X 0,Y 186.886,Z 528.284,A -85,B 0,C 180,E1 -23629.903,E2 -23629.903} C_VEL
LIN {X 0,Y 184.568,Z 541.051,A -85,B 0,C 180,E1 -23631.076,E2 -23631.076} C_VEL
LIN {X 0,Y 181.855,Z 552.34,A -85,B 0,C 180,E1 -23632.506,E2 -23632.506} C_VEL
LIN {X 0,Y 178.395,Z 563.967,A -85,B 0,C 180,E1 -23634.473,E2 -23634.473} C_VEL
LIN {X 0,Y 174.784,Z 574.41,A -85,B 0,C 180,E1 -23636.78,E2 -23636.78} C_VEL
LIN {X 0,Y 171.431,Z 582.947,A -85,B 0,C 180,E1 -23639.174,E2 -23639.174} C_VEL
LIN {X 0,Y 168.095,Z 590.967,A -85,B 0,C 180,E1 -23642.019,E2 -23642.019} C_VEL
LIN {X 0,Y 164.514,Z 598.483,A -85,B 0,C 180,E1 -23645.385,E2 -23645.385} C_VEL
LIN {X 0,Y 160.948,Z 605.538,A -85,B 0,C 180,E1 -23649.554,E2 -23649.554} C_VEL
LIN {X 0,Y 158.62,Z 610.231,A -85,B 0,C 180,E1 -23653.262,E2 -23653.262} C_VEL
LIN {X 0,Y 156.854,Z 613.82,A -85,B 0,C 180,E1 -23657.055,E2 -23657.055} C_VEL
LIN {X 0,Y 156.017,Z 615.672,A -85,B 0,C 180,E1 -23659.62,E2 -23659.62} C_VEL
LIN {X 0,Y 155.026,Z 618.05,A -85,B 0,C 180,E1 -23664.798,E2 -23664.798} C_VEL
LIN {X 0,Y 154.845,Z 618.656,A -85,B 0,C 180,E1 -23667.399,E2 -23667.399} C_VEL
LIN {X 0,Y 154.794,Z 618.883,A -85,B 0,C 180,E1 -23670,E2 -23670} C_VEL
LIN {X 0,Y 154.869,Z 618.565,A -85,B 0,C 180,E1 -23673.269,E2 -23673.269} C_VEL
LIN {X 0,Y 155.36,Z 617.133,A -85,B 0,C 180,E1 -23677.8,E2 -23677.8} C_VEL
LIN {X 0,Y 156.019,Z 615.772,A -85,B 0,C 180,E1 -23680.381,E2 -23680.381} C_VEL
LIN {X 0,Y 157.368,Z 612.9,A -85,B 0,C 180,E1 -23684.22,E2 -23684.22} C_VEL
LIN {X 0,Y 159.304,Z 609.002,A -85,B 0,C 180,E1 -23687.989,E2 -23687.989} C_VEL
LIN {X 0,Y 161.834,Z 603.973,A -85,B 0,C 180,E1 -23691.663,E2 -23691.663} C_VEL
LIN {X 0,Y 165.049,Z 597.635,A -85,B 0,C 180,E1 -23695.203,E2 -23695.203} C_VEL
LIN {X 0,Y 168.324,Z 590.45,A -85,B 0,C 180,E1 -23698.356,E2 -23698.356} C_VEL
LIN {X 0,Y 172.039,Z 581.63,A -85,B 0,C 180,E1 -23701.39,E2 -23701.39} C_VEL
LIN {X 0,Y 175.812,Z 571.767,A -85,B 0,C 180,E1 -23704.032,E2 -23704.032} C_VEL
LIN {X 0,Y 179.59,Z 560.652,A -85,B 0,C 180,E1 -23706.292,E2 -23706.292} C_VEL
LIN {X 0,Y 182.71,Z 549.756,A -85,B 0,C 180,E1 -23707.985,E2 -23707.985} C_VEL
LIN {X 0,Y 185.428,Z 537.709,A -85,B 0,C 180,E1 -23709.41,E2 -23709.41} C_VEL
LIN {X 0,Y 187.535,Z 525.072,A -85,B 0,C 180,E1 -23710.472,E2 -23710.472} C_VEL
LIN {X 0,Y 189.017,Z 511.469,A -85,B 0,C 180,E1 -23711.171,E2 -23711.171} C_VEL
LIN {X 0,Y 191.499,Z 470.584,A -85,B 0,C 180,E1 -23712.554,E2 -23712.554} C_VEL
LIN {X 0,Y 185.872,Z 457.247,A -85,B 0,C 180,E1 -23714.885,E2 -23714.885} C_VEL
LIN {X 0,Y 182.535,Z 450.825,A -85,B 0,C 180,E1 -23716.302,E2 -23716.302} C_VEL
LIN {X 0,Y 176.234,Z 440.737,A -85,B 0,C 180,E1 -23719.114,E2 -23719.114} C_VEL
LIN {X 0,Y 171.083,Z 433.225,A -85,B 0,C 180,E1 -23721.656,E2 -23721.656} C_VEL
LIN {X 0,Y 168.111,Z 429.136,A -85,B 0,C 180,E1 -23723.248,E2 -23723.248} C_VEL
LIN {X 0,Y 165.427,Z 425.341,A -85,B 0,C 180,E1 -23724.799,E2 -23724.799} C_VEL
LIN {X 0,Y 162.413,Z 421.996,A -85,B 0,C 180,E1 -23726.607,E2 -23726.607} C_VEL
LIN {X 0,Y 161.319,Z 419.889,A -85,B 0,C 180,E1 -23727.375,E2 -23727.375} C_VEL
LIN {X 0,Y 158.997,Z 418.097,A -85,B 0,C 180,E1 -23728.868,E2 -23728.868} C_VEL
LIN {X 0,Y 157.643,Z 415.854,A -85,B 0,C 180,E1 -23729.897,E2 -23729.897} C_VEL
LIN {X 0,Y 157.3,Z 414.38,A -85,B 0,C 180,E1 -23730.379,E2 -23730.379} C_VEL
LIN {X 0,Y 157.326,Z 414.384,A -85,B 0,C 180,E1 -23733.467,E2 -23733.467} C_VEL
LIN {X 0,Y 157.45,Z 414.36,A -85,B 0,C 180,E1 -23739.616,E2 -23739.616} C_VEL
LIN {X 0,Y 157.492,Z 414.363,A -85,B 0,C 180,E1 -23744.47,E2 -23744.47} C_VEL
LIN {X 0,Y 157.775,Z 414.333,A -85,B 0,C 180,E1 -23749.736,E2 -23749.736} C_VEL
LIN {X 0,Y 157.826,Z 414.308,A -85,B 0,C 180,E1 -23752.323,E2 -23752.323} C_VEL
LIN {X 0,Y 158.262,Z 414.255,A -85,B 0,C 180,E1 -23760,E2 -23760} C_VEL
LIN {X 0,Y 157.77,Z 414.328,A -85,B 0,C 180,E1 -23767.68,E2 -23767.68} C_VEL
LIN {X 0,Y 157.64,Z 414.333,A -85,B 0,C 180,E1 -23771.237,E2 -23771.237} C_VEL
LIN {X 0,Y 157.457,Z 414.366,A -85,B 0,C 180,E1 -23775.534,E2 -23775.534} C_VEL
LIN {X 0,Y 157.373,Z 414.376,A -85,B 0,C 180,E1 -23780.932,E2 -23780.932} C_VEL
LIN {X 0,Y 157.317,Z 414.388,A -85,B 0,C 180,E1 -23786.684,E2 -23786.684} C_VEL
LIN {X 0,Y 157.282,Z 414.393,A -85,B 0,C 180,E1 -23789.441,E2 -23789.441} C_VEL
LIN {X 0,Y 158.1,Z 416.848,A -85,B 0,C 180,E1 -23790.19,E2 -23790.19} C_VEL
LIN {X 0,Y 160.127,Z 419.198,A -85,B 0,C 180,E1 -23791.605,E2 -23791.605} C_VEL
LIN {X 0,Y 161.524,Z 420.293,A -85,B 0,C 180,E1 -23792.485,E2 -23792.485} C_VEL
LIN {X 0,Y 163.486,Z 423.482,A -85,B 0,C 180,E1 -23793.791,E2 -23793.791} C_VEL
LIN {X 0,Y 165.37,Z 425.329,A -85,B 0,C 180,E1 -23794.886,E2 -23794.886} C_VEL
LIN {X 0,Y 168.806,Z 430.189,A -85,B 0,C 180,E1 -23796.855,E2 -23796.855} C_VEL
LIN {X 0,Y 174.647,Z 439.828,A -85,B 0,C 180,E1 -23799.935,E2 -23799.935} C_VEL
LIN {X 0,Y 181.054,Z 451.919,A -85,B 0,C 180,E1 -23802.979,E2 -23802.979} C_VEL
LIN {X 0,Y 186.491,Z 463.947,A -85,B 0,C 180,E1 -23805.374,E2 -23805.374} C_VEL
LIN {X 0,Y 191.02,Z 475.64,A -85,B 0,C 180,E1 -23807.281,E2 -23807.281} C_VEL
LIN {X 0,Y 190.791,Z 483.365,A -85,B 0,C 180,E1 -23807.604,E2 -23807.604} C_VEL
LIN {X 0,Y 188.274,Z 522.058,A -85,B 0,C 180,E1 -23808.921,E2 -23808.921} C_VEL
LIN {X 0,Y 186.458,Z 535.862,A -85,B 0,C 180,E1 -23809.754,E2 -23809.754} C_VEL
LIN {X 0,Y 183.946,Z 548.645,A -85,B 0,C 180,E1 -23810.919,E2 -23810.919} C_VEL
LIN {X 0,Y 180.613,Z 561.304,A -85,B 0,C 180,E1 -23812.554,E2 -23812.554} C_VEL
LIN {X 0,Y 177.096,Z 572.567,A -85,B 0,C 180,E1 -23814.521,E2 -23814.521} C_VEL
LIN {X 0,Y 173.323,Z 582.711,A -85,B 0,C 180,E1 -23816.81,E2 -23816.81} C_VEL
LIN {X 0,Y 169.538,Z 591.852,A -85,B 0,C 180,E1 -23819.481,E2 -23819.481} C_VEL
LIN {X 0,Y 167.185,Z 597.247,A -85,B 0,C 180,E1 -23821.412,E2 -23821.412} C_VEL
LIN {X 0,Y 164.989,Z 600.922,A -85,B 0,C 180,E1 -23822.816,E2 -23822.816} C_VEL
LIN {X 0,Y 159.816,Z 606.408,A -85,B 0,C 180,E1 -23825.086,E2 -23825.086} C_VEL
LIN {X 0,Y 154.703,Z 611.286,A -85,B 0,C 180,E1 -23827.642,E2 -23827.642} C_VEL
LIN {X 0,Y 152.662,Z 613.907,A -85,B 0,C 180,E1 -23829.463,E2 -23829.463} C_VEL
LIN {X 0,Y 150.195,Z 618.637,A -85,B 0,C 180,E1 -23833.694,E2 -23833.694} C_VEL
LIN {X 0,Y 149.183,Z 620.932,A -85,B 0,C 180,E1 -23836.375,E2 -23836.375} C_VEL
LIN {X 0,Y 148.407,Z 622.79,A -85,B 0,C 180,E1 -23839.08,E2 -23839.08} C_VEL
LIN {X 0,Y 147.902,Z 624.184,A -85,B 0,C 180,E1 -23841.804,E2 -23841.804} C_VEL
LIN {X 0,Y 147.626,Z 625.181,A -85,B 0,C 180,E1 -23844.536,E2 -23844.536} C_VEL
LIN {X 0,Y 147.606,Z 625.959,A -85,B 0,C 180,E1 -23849.109,E2 -23849.109} C_VEL
LIN {X 0,Y 147.569,Z 625.776,A -85,B 0,C 180,E1 -23852.729,E2 -23852.729} C_VEL
LIN {X 0,Y 147.635,Z 625.158,A -85,B 0,C 180,E1 -23855.463,E2 -23855.463} C_VEL
LIN {X 0,Y 147.902,Z 624.152,A -85,B 0,C 180,E1 -23858.195,E2 -23858.195} C_VEL
LIN {X 0,Y 148.407,Z 622.743,A -85,B 0,C 180,E1 -23860.919,E2 -23860.919} C_VEL
LIN {X 0,Y 149.67,Z 619.792,A -85,B 0,C 180,E1 -23864.967,E2 -23864.967} C_VEL
LIN {X 0,Y 151.599,Z 615.805,A -85,B 0,C 180,E1 -23868.936,E2 -23868.936} C_VEL
LIN {X 0,Y 154.752,Z 609.68,A -85,B 0,C 180,E1 -23873.414,E2 -23873.414} C_VEL
LIN {X 0,Y 157.578,Z 604.233,A -85,B 0,C 180,E1 -23876.487,E2 -23876.487} C_VEL
LIN {X 0,Y 161.275,Z 596.192,A -85,B 0,C 180,E1 -23880.075,E2 -23880.075} C_VEL
LIN {X 0,Y 164.973,Z 588.003,A -85,B 0,C 180,E1 -23882.899,E2 -23882.899} C_VEL
LIN {X 0,Y 169.1,Z 578.017,A -85,B 0,C 180,E1 -23885.581,E2 -23885.581} C_VEL
LIN {X 0,Y 173.164,Z 566.727,A -85,B 0,C 180,E1 -23887.869,E2 -23887.869} C_VEL
LIN {X 0,Y 176.494,Z 555.663,A -85,B 0,C 180,E1 -23889.577,E2 -23889.577} C_VEL
LIN {X 0,Y 179.488,Z 543.381,A -85,B 0,C 180,E1 -23890.985,E2 -23890.985} C_VEL
LIN {X 0,Y 181.902,Z 530.074,A -85,B 0,C 180,E1 -23892.013,E2 -23892.013} C_VEL
LIN {X 0,Y 183.382,Z 516.282,A -85,B 0,C 180,E1 -23892.69,E2 -23892.69} C_VEL
LIN {X 0,Y 185.7,Z 477.972,A -85,B 0,C 180,E1 -23894.022,E2 -23894.022} C_VEL
LIN {X 0,Y 181.262,Z 466.313,A -85,B 0,C 180,E1 -23896.031,E2 -23896.031} C_VEL
LIN {X 0,Y 176.769,Z 456.185,A -85,B 0,C 180,E1 -23898.149,E2 -23898.149} C_VEL
LIN {X 0,Y 171.551,Z 446.076,A -85,B 0,C 180,E1 -23900.769,E2 -23900.769} C_VEL
LIN {X 0,Y 166.816,Z 437.893,A -85,B 0,C 180,E1 -23903.363,E2 -23903.363} C_VEL
LIN {X 0,Y 164.535,Z 434.312,A -85,B 0,C 180,E1 -23904.701,E2 -23904.701} C_VEL
LIN {X 0,Y 161.811,Z 430.499,A -85,B 0,C 180,E1 -23906.374,E2 -23906.374} C_VEL
LIN {X 0,Y 159.276,Z 427.253,A -85,B 0,C 180,E1 -23908.029,E2 -23908.029} C_VEL
LIN {X 0,Y 158.349,Z 425.955,A -85,B 0,C 180,E1 -23908.676,E2 -23908.676} C_VEL
LIN {X 0,Y 155.853,Z 423.286,A -85,B 0,C 180,E1 -23910.448,E2 -23910.448} C_VEL
LIN {X 0,Y 154.602,Z 420.964,A -85,B 0,C 180,E1 -23911.49,E2 -23911.49} C_VEL
LIN {X 0,Y 152.199,Z 419.306,A -85,B 0,C 180,E1 -23913.357,E2 -23913.357} C_VEL
LIN {X 0,Y 150.671,Z 416.953,A -85,B 0,C 180,E1 -23914.785,E2 -23914.785} C_VEL
LIN {X 0,Y 150.241,Z 415.264,A -85,B 0,C 180,E1 -23915.379,E2 -23915.379} C_VEL
LIN {X 0,Y 150.394,Z 415.241,A -85,B 0,C 180,E1 -23920.906,E2 -23920.906} C_VEL
LIN {X 0,Y 150.44,Z 415.238,A -85,B 0,C 180,E1 -23926.492,E2 -23926.492} C_VEL
LIN {X 0,Y 150.612,Z 415.216,A -85,B 0,C 180,E1 -23929.243,E2 -23929.243} C_VEL
LIN {X 0,Y 150.705,Z 415.208,A -85,B 0,C 180,E1 -23931.958,E2 -23931.958} C_VEL
LIN {X 0,Y 151.219,Z 415.138,A -85,B 0,C 180,E1 -23940,E2 -23940} C_VEL
LIN {X 0,Y 150.765,Z 415.199,A -85,B 0,C 180,E1 -23948.039,E2 -23948.039} C_VEL
LIN {X 0,Y 150.636,Z 415.209,A -85,B 0,C 180,E1 -23951.547,E2 -23951.547} C_VEL
LIN {X 0,Y 150.397,Z 415.24,A -85,B 0,C 180,E1 -23956.283,E2 -23956.283} C_VEL
LIN {X 0,Y 150.391,Z 415.244,A -85,B 0,C 180,E1 -23960.832,E2 -23960.832} C_VEL
LIN {X 0,Y 150.267,Z 415.376,A -85,B 0,C 180,E1 -23965.091,E2 -23965.091} C_VEL
LIN {X 0,Y 150.9,Z 417.482,A -85,B 0,C 180,E1 -23965.831,E2 -23965.831} C_VEL
LIN {X 0,Y 152.821,Z 419.902,A -85,B 0,C 180,E1 -23967.536,E2 -23967.536} C_VEL
LIN {X 0,Y 154.875,Z 421.33,A -85,B 0,C 180,E1 -23969.105,E2 -23969.105} C_VEL
LIN {X 0,Y 156.669,Z 424.412,A -85,B 0,C 180,E1 -23970.546,E2 -23970.546} C_VEL
LIN {X 0,Y 158.986,Z 426.656,A -85,B 0,C 180,E1 -23972.131,E2 -23972.131} C_VEL
LIN {X 0,Y 161.474,Z 430.194,A -85,B 0,C 180,E1 -23973.8,E2 -23973.8} C_VEL
LIN {X 0,Y 162.836,Z 431.811,A -85,B 0,C 180,E1 -23974.638,E2 -23974.638} C_VEL
LIN {X 0,Y 166.598,Z 437.11,A -85,B 0,C 180,E1 -23976.857,E2 -23976.857} C_VEL
LIN {X 0,Y 171.82,Z 444.745,A -85,B 0,C 180,E1 -23979.631,E2 -23979.631} C_VEL
LIN {X 0,Y 178.077,Z 454.92,A -85,B 0,C 180,E1 -23982.617,E2 -23982.617} C_VEL
LIN {X 0,Y 181.282,Z 461.08,A -85,B 0,C 180,E1 -23984.06,E2 -23984.06} C_VEL
LIN {X 0,Y 186.025,Z 472.629,A -85,B 0,C 180,E1 -23986.17,E2 -23986.17} C_VEL
LIN {X 0,Y 183.201,Z 515.864,A -85,B 0,C 180,E1 -23987.693,E2 -23987.693} C_VEL
LIN {X 0,Y 181.408,Z 529.07,A -85,B 0,C 180,E1 -23988.504,E2 -23988.504} C_VEL
LIN {X 0,Y 179.109,Z 541.225,A -85,B 0,C 180,E1 -23989.652,E2 -23989.652} C_VEL
LIN {X 0,Y 176.28,Z 552.513,A -85,B 0,C 180,E1 -23991.103,E2 -23991.103} C_VEL
LIN {X 0,Y 172.674,Z 564.138,A -85,B 0,C 180,E1 -23993.106,E2 -23993.106} C_VEL
LIN {X 0,Y 168.89,Z 574.581,A -85,B 0,C 180,E1 -23995.461,E2 -23995.461} C_VEL
LIN {X 0,Y 165.359,Z 583.117,A -85,B 0,C 180,E1 -23997.911,E2 -23997.911} C_VEL
LIN {X 0,Y 161.791,Z 591.264,A -85,B 0,C 180,E1 -24000.889,E2 -24000.889} C_VEL
LIN {X 0,Y 158.092,Z 598.652,A -85,B 0,C 180,E1 -24004.315,E2 -24004.315} C_VEL
LIN {X 0,Y 154.302,Z 605.707,A -85,B 0,C 180,E1 -24008.631,E2 -24008.631} C_VEL
LIN {X 0,Y 151.833,Z 610.399,A -85,B 0,C 180,E1 -24012.491,E2 -24012.491} C_VEL
LIN {X 0,Y 149.947,Z 613.988,A -85,B 0,C 180,E1 -24016.447,E2 -24016.447} C_VEL
LIN {X 0,Y 149.032,Z 615.839,A -85,B 0,C 180,E1 -24019.128,E2 -24019.128} C_VEL
LIN {X 0,Y 147.949,Z 618.218,A -85,B 0,C 180,E1 -24024.549,E2 -24024.549} C_VEL
LIN {X 0,Y 147.756,Z 618.823,A -85,B 0,C 180,E1 -24027.274,E2 -24027.274} C_VEL
LIN {X 0,Y 147.718,Z 619.049,A -85,B 0,C 180,E1 -24030.001,E2 -24030.001} C_VEL
LIN {X 0,Y 147.756,Z 618.854,A -85,B 0,C 180,E1 -24032.727,E2 -24032.727} C_VEL
LIN {X 0,Y 147.949,Z 618.268,A -85,B 0,C 180,E1 -24035.452,E2 -24035.452} C_VEL
LIN {X 0,Y 149.034,Z 615.939,A -85,B 0,C 180,E1 -24040.873,E2 -24040.873} C_VEL
LIN {X 0,Y 150.484,Z 613.066,A -85,B 0,C 180,E1 -24044.885,E2 -24044.885} C_VEL
LIN {X 0,Y 152.555,Z 609.168,A -85,B 0,C 180,E1 -24048.814,E2 -24048.814} C_VEL
LIN {X 0,Y 155.247,Z 604.139,A -85,B 0,C 180,E1 -24052.632,E2 -24052.632} C_VEL
LIN {X 0,Y 158.649,Z 597.8,A -85,B 0,C 180,E1 -24056.295,E2 -24056.295} C_VEL
LIN {X 0,Y 162.675,Z 589.391,A -85,B 0,C 180,E1 -24060.025,E2 -24060.025} C_VEL
LIN {X 0,Y 166.777,Z 580.016,A -85,B 0,C 180,E1 -24063.218,E2 -24063.218} C_VEL
LIN {X 0,Y 170.889,Z 569.653,A -85,B 0,C 180,E1 -24065.878,E2 -24065.878} C_VEL
LIN {X 0,Y 174.833,Z 557.969,A -85,B 0,C 180,E1 -24068.175,E2 -24068.175} C_VEL
LIN {X 0,Y 178.11,Z 546.297,A -85,B 0,C 180,E1 -24069.883,E2 -24069.883} C_VEL
LIN {X 0,Y 180.727,Z 534.152,A -85,B 0,C 180,E1 -24071.198,E2 -24071.198} C_VEL
LIN {X 0,Y 182.787,Z 520.816,A -85,B 0,C 180,E1 -24072.201,E2 -24072.201} C_VEL
LIN {X 0,Y 184.095,Z 506.996,A -85,B 0,C 180,E1 -24072.787,E2 -24072.787} C_VEL
LIN {X 0,Y 186.194,Z 472.733,A -85,B 0,C 180,E1 -24073.966,E2 -24073.966} C_VEL
LIN {X 0,Y 181.081,Z 460.465,A -85,B 0,C 180,E1 -24076.242,E2 -24076.242} C_VEL
LIN {X 0,Y 177.089,Z 453.118,A -85,B 0,C 180,E1 -24078.051,E2 -24078.051} C_VEL
LIN {X 0,Y 170.684,Z 442.904,A -85,B 0,C 180,E1 -24081.184,E2 -24081.184} C_VEL
LIN {X 0,Y 165.198,Z 434.967,A -85,B 0,C 180,E1 -24084.203,E2 -24084.203} C_VEL
LIN {X 0,Y 161.897,Z 430.587,A -85,B 0,C 180,E1 -24086.207,E2 -24086.207} C_VEL
LIN {X 0,Y 159.177,Z 427.012,A -85,B 0,C 180,E1 -24088.006,E2 -24088.006} C_VEL
LIN {X 0,Y 158.407,Z 425.987,A -85,B 0,C 180,E1 -24088.545,E2 -24088.545} C_VEL
LIN {X 0,Y 155.966,Z 423.408,A -85,B 0,C 180,E1 -24090.286,E2 -24090.286} C_VEL
LIN {X 0,Y 154.529,Z 420.941,A -85,B 0,C 180,E1 -24091.475,E2 -24091.475} C_VEL
LIN {X 0,Y 152.033,Z 419.104,A -85,B 0,C 180,E1 -24093.458,E2 -24093.458} C_VEL
LIN {X 0,Y 150.597,Z 416.78,A -85,B 0,C 180,E1 -24094.837,E2 -24094.837} C_VEL
LIN {X 0,Y 150.248,Z 415.255,A -85,B 0,C 180,E1 -24095.38,E2 -24095.38} C_VEL
LIN {X 0,Y 150.404,Z 415.234,A -85,B 0,C 180,E1 -24100.907,E2 -24100.907} C_VEL
LIN {X 0,Y 150.471,Z 415.224,A -85,B 0,C 180,E1 -24106.495,E2 -24106.495} C_VEL
LIN {X 0,Y 150.692,Z 415.214,A -85,B 0,C 180,E1 -24109.248,E2 -24109.248} C_VEL
LIN {X 0,Y 150.765,Z 415.188,A -85,B 0,C 180,E1 -24111.961,E2 -24111.961} C_VEL
LIN {X 0,Y 151.222,Z 415.131,A -85,B 0,C 180,E1 -24120,E2 -24120} C_VEL
LIN {X 0,Y 150.708,Z 415.21,A -85,B 0,C 180,E1 -24128.042,E2 -24128.042} C_VEL
LIN {X 0,Y 150.581,Z 415.211,A -85,B 0,C 180,E1 -24131.438,E2 -24131.438} C_VEL
LIN {X 0,Y 150.364,Z 415.242,A -85,B 0,C 180,E1 -24136.286,E2 -24136.286} C_VEL
LIN {X 0,Y 150.354,Z 415.25,A -85,B 0,C 180,E1 -24140.792,E2 -24140.792} C_VEL
LIN {X 0,Y 150.254,Z 415.35,A -85,B 0,C 180,E1 -24144.435,E2 -24144.435} C_VEL
LIN {X 0,Y 150.986,Z 417.681,A -85,B 0,C 180,E1 -24145.29,E2 -24145.29} C_VEL
LIN {X 0,Y 153.06,Z 420.093,A -85,B 0,C 180,E1 -24147.119,E2 -24147.119} C_VEL
LIN {X 0,Y 154.815,Z 421.29,A -85,B 0,C 180,E1 -24148.467,E2 -24148.467} C_VEL
LIN {X 0,Y 156.696,Z 424.405,A -85,B 0,C 180,E1 -24149.984,E2 -24149.984} C_VEL
LIN {X 0,Y 159.014,Z 426.675,A -85,B 0,C 180,E1 -24151.585,E2 -24151.585} C_VEL
LIN {X 0,Y 161.246,Z 429.927,A -85,B 0,C 180,E1 -24153.105,E2 -24153.105} C_VEL
LIN {X 0,Y 162.879,Z 431.868,A -85,B 0,C 180,E1 -24154.12,E2 -24154.12} C_VEL
LIN {X 0,Y 166.336,Z 437.002,A -85,B 0,C 180,E1 -24156.199,E2 -24156.199} C_VEL
LIN {X 0,Y 171.251,Z 445.393,A -85,B 0,C 180,E1 -24158.929,E2 -24158.929} C_VEL
LIN {X 0,Y 177.18,Z 456.932,A -85,B 0,C 180,E1 -24161.922,E2 -24161.922} C_VEL
LIN {X 0,Y 182.417,Z 468.961,A -85,B 0,C 180,E1 -24164.38,E2 -24164.38} C_VEL
LIN {X 0,Y 185.851,Z 478.127,A -85,B 0,C 180,E1 -24165.93,E2 -24165.93} C_VEL
LIN {X 0,Y 183.001,Z 521.906,A -85,B 0,C 180,E1 -24167.465,E2 -24167.465} C_VEL
LIN {X 0,Y 181.153,Z 535.457,A -85,B 0,C 180,E1 -24168.288,E2 -24168.288} C_VEL
LIN {X 0,Y 178.501,Z 548.485,A -85,B 0,C 180,E1 -24169.484,E2 -24169.484} C_VEL
LIN {X 0,Y 175.016,Z 561.141,A -85,B 0,C 180,E1 -24171.138,E2 -24171.138} C_VEL
LIN {X 0,Y 171.349,Z 572.404,A -85,B 0,C 180,E1 -24173.14,E2 -24173.14} C_VEL
LIN {X 0,Y 167.434,Z 582.547,A -85,B 0,C 180,E1 -24175.482,E2 -24175.482} C_VEL
LIN {X 0,Y 163.451,Z 591.688,A -85,B 0,C 180,E1 -24178.215,E2 -24178.215} C_VEL
LIN {X 0,Y 159.27,Z 600.73,A -85,B 0,C 180,E1 -24181.748,E2 -24181.748} C_VEL
LIN {X 0,Y 155.864,Z 607.779,A -85,B 0,C 180,E1 -24185.348,E2 -24185.348} C_VEL
LIN {X 0,Y 152.662,Z 613.907,A -85,B 0,C 180,E1 -24189.463,E2 -24189.463} C_VEL
LIN {X 0,Y 150.745,Z 616.332,A -85,B 0,C 180,E1 -24191.371,E2 -24191.371} C_VEL
LIN {X 0,Y 146.257,Z 619.668,A -85,B 0,C 180,E1 -24194.535,E2 -24194.535} C_VEL
LIN {X 0,Y 142.866,Z 621.79,A -85,B 0,C 180,E1 -24197.26,E2 -24197.26} C_VEL
LIN {X 0,Y 141.267,Z 623.121,A -85,B 0,C 180,E1 -24199.497,E2 -24199.497} C_VEL
LIN {X 0,Y 141.032,Z 623.474,A -85,B 0,C 180,E1 -24200.275,E2 -24200.275} C_VEL
LIN {X 0,Y 140.55,Z 625.014,A -85,B 0,C 180,E1 -24204.26,E2 -24204.26} C_VEL
LIN {X 0,Y 140.486,Z 625.624,A -85,B 0,C 180,E1 -24207.132,E2 -24207.132} C_VEL
LIN {X 0,Y 140.56,Z 625.837,A -85,B 0,C 180,E1 -24209.999,E2 -24209.999} C_VEL
LIN {X 0,Y 140.487,Z 625.609,A -85,B 0,C 180,E1 -24212.867,E2 -24212.867} C_VEL
LIN {X 0,Y 140.555,Z 624.99,A -85,B 0,C 180,E1 -24215.739,E2 -24215.739} C_VEL
LIN {X 0,Y 140.853,Z 623.984,A -85,B 0,C 180,E1 -24218.608,E2 -24218.608} C_VEL
LIN {X 0,Y 141.418,Z 622.574,A -85,B 0,C 180,E1 -24221.466,E2 -24221.466} C_VEL
LIN {X 0,Y 142.796,Z 619.623,A -85,B 0,C 180,E1 -24225.705,E2 -24225.705} C_VEL
LIN {X 0,Y 144.893,Z 615.637,A -85,B 0,C 180,E1 -24229.848,E2 -24229.848} C_VEL
LIN {X 0,Y 148.236,Z 609.511,A -85,B 0,C 180,E1 -24234.509,E2 -24234.509} C_VEL
LIN {X 0,Y 151.182,Z 604.062,A -85,B 0,C 180,E1 -24237.701,E2 -24237.701} C_VEL
LIN {X 0,Y 155.15,Z 596.022,A -85,B 0,C 180,E1 -24241.394,E2 -24241.394} C_VEL
LIN {X 0,Y 159.06,Z 587.833,A -85,B 0,C 180,E1 -24244.288,E2 -24244.288} C_VEL
LIN {X 0,Y 163.381,Z 577.847,A -85,B 0,C 180,E1 -24247.029,E2 -24247.029} C_VEL
LIN {X 0,Y 167.617,Z 566.556,A -85,B 0,C 180,E1 -24249.358,E2 -24249.358} C_VEL
LIN {X 0,Y 171.08,Z 555.49,A -85,B 0,C 180,E1 -24251.093,E2 -24251.093} C_VEL
LIN {X 0,Y 174.199,Z 543.207,A -85,B 0,C 180,E1 -24252.514,E2 -24252.514} C_VEL
LIN {X 0,Y 176.596,Z 530.586,A -85,B 0,C 180,E1 -24253.509,E2 -24253.509} C_VEL
LIN {X 0,Y 178.13,Z 517.193,A -85,B 0,C 180,E1 -24254.196,E2 -24254.196} C_VEL
LIN {X 0,Y 180.516,Z 480.032,A -85,B 0,C 180,E1 -24255.509,E2 -24255.509} C_VEL
LIN {X 0,Y 176.223,Z 468.678,A -85,B 0,C 180,E1 -24257.605,E2 -24257.605} C_VEL
LIN {X 0,Y 172.436,Z 460.133,A -85,B 0,C 180,E1 -24259.524,E2 -24259.524} C_VEL
LIN {X 0,Y 167.915,Z 451.058,A -85,B 0,C 180,E1 -24261.965,E2 -24261.965} C_VEL
LIN {X 0,Y 163.961,Z 444.009,A -85,B 0,C 180,E1 -24264.267,E2 -24264.267} C_VEL
LIN {X 0,Y 161.578,Z 440.042,A -85,B 0,C 180,E1 -24265.755,E2 -24265.755} C_VEL
LIN {X 0,Y 159.03,Z 436.44,A -85,B 0,C 180,E1 -24267.411,E2 -24267.411} C_VEL
LIN {X 0,Y 156.371,Z 432.712,A -85,B 0,C 180,E1 -24269.282,E2 -24269.282} C_VEL
LIN {X 0,Y 153.164,Z 428.921,A -85,B 0,C 180,E1 -24271.712,E2 -24271.712} C_VEL
LIN {X 0,Y 152.243,Z 427.412,A -85,B 0,C 180,E1 -24272.508,E2 -24272.508} C_VEL
LIN {X 0,Y 149.519,Z 424.911,A -85,B 0,C 180,E1 -24274.842,E2 -24274.842} C_VEL
LIN {X 0,Y 147.903,Z 421.922,A -85,B 0,C 180,E1 -24276.549,E2 -24276.549} C_VEL
LIN {X 0,Y 145.507,Z 420.385,A -85,B 0,C 180,E1 -24279.012,E2 -24279.012} C_VEL
LIN {X 0,Y 143.865,Z 418.045,A -85,B 0,C 180,E1 -24281.117,E2 -24281.117} C_VEL
LIN {X 0,Y 143.309,Z 416.13,A -85,B 0,C 180,E1 -24282.151,E2 -24282.151} C_VEL
LIN {X 0,Y 143.538,Z 416.1,A -85,B 0,C 180,E1 -24288.706,E2 -24288.706} C_VEL
LIN {X 0,Y 143.626,Z 416.086,A -85,B 0,C 180,E1 -24291.559,E2 -24291.559} C_VEL
LIN {X 0,Y 144.178,Z 416.014,A -85,B 0,C 180,E1 -24300,E2 -24300} C_VEL
LIN {X 0,Y 143.686,Z 416.083,A -85,B 0,C 180,E1 -24308.438,E2 -24308.438} C_VEL
LIN {X 0,Y 143.572,Z 416.088,A -85,B 0,C 180,E1 -24311.758,E2 -24311.758} C_VEL
LIN {X 0,Y 143.36,Z 416.318,A -85,B 0,C 180,E1 -24318.397,E2 -24318.397} C_VEL
LIN {X 0,Y 144.275,Z 418.871,A -85,B 0,C 180,E1 -24319.845,E2 -24319.845} C_VEL
LIN {X 0,Y 146.593,Z 421.329,A -85,B 0,C 180,E1 -24322.553,E2 -24322.553} C_VEL
LIN {X 0,Y 148.126,Z 422.265,A -85,B 0,C 180,E1 -24324.063,E2 -24324.063} C_VEL
LIN {X 0,Y 149.891,Z 425.389,A -85,B 0,C 180,E1 -24325.885,E2 -24325.885} C_VEL
LIN {X 0,Y 152.602,Z 427.853,A -85,B 0,C 180,E1 -24328.168,E2 -24328.168} C_VEL
LIN {X 0,Y 155.016,Z 431.389,A -85,B 0,C 180,E1 -24330.127,E2 -24330.127} C_VEL
LIN {X 0,Y 156.599,Z 433.1,A -85,B 0,C 180,E1 -24331.267,E2 -24331.267} C_VEL
LIN {X 0,Y 159.407,Z 436.834,A -85,B 0,C 180,E1 -24333.207,E2 -24333.207} C_VEL
LIN {X 0,Y 163.617,Z 442.891,A -85,B 0,C 180,E1 -24335.86,E2 -24335.86} C_VEL
LIN {X 0,Y 168.408,Z 450.149,A -85,B 0,C 180,E1 -24338.563,E2 -24338.563} C_VEL
LIN {X 0,Y 174.198,Z 459.741,A -85,B 0,C 180,E1 -24341.498,E2 -24341.498} C_VEL
LIN {X 0,Y 177.368,Z 466.089,A -85,B 0,C 180,E1 -24343.022,E2 -24343.022} C_VEL
LIN {X 0,Y 180.846,Z 474.822,A -85,B 0,C 180,E1 -24344.684,E2 -24344.684} C_VEL
LIN {X 0,Y 178.096,Z 515.288,A -85,B 0,C 180,E1 -24346.115,E2 -24346.115} C_VEL
LIN {X 0,Y 176.268,Z 528.647,A -85,B 0,C 180,E1 -24346.932,E2 -24346.932} C_VEL
LIN {X 0,Y 173.758,Z 541.399,A -85,B 0,C 180,E1 -24348.136,E2 -24348.136} C_VEL
LIN {X 0,Y 170.819,Z 552.685,A -85,B 0,C 180,E1 -24349.609,E2 -24349.609} C_VEL
LIN {X 0,Y 167.064,Z 564.309,A -85,B 0,C 180,E1 -24351.648,E2 -24351.648} C_VEL
LIN {X 0,Y 163.079,Z 574.752,A -85,B 0,C 180,E1 -24354.043,E2 -24354.043} C_VEL
LIN {X 0,Y 159.382,Z 583.284,A -85,B 0,C 180,E1 -24356.552,E2 -24356.552} C_VEL
LIN {X 0,Y 155.044,Z 592.525,A -85,B 0,C 180,E1 -24360.092,E2 -24360.092} C_VEL
LIN {X 0,Y 151.101,Z 599.932,A -85,B 0,C 180,E1 -24363.778,E2 -24363.778} C_VEL
LIN {X 0,Y 147.701,Z 605.876,A -85,B 0,C 180,E1 -24367.626,E2 -24367.626} C_VEL
LIN {X 0,Y 145.061,Z 610.568,A -85,B 0,C 180,E1 -24371.645,E2 -24371.645} C_VEL
LIN {X 0,Y 143.037,Z 614.156,A -85,B 0,C 180,E1 -24375.779,E2 -24375.779} C_VEL
LIN {X 0,Y 142.053,Z 616.008,A -85,B 0,C 180,E1 -24378.586,E2 -24378.586} C_VEL
LIN {X 0,Y 140.876,Z 618.385,A -85,B 0,C 180,E1 -24384.274,E2 -24384.274} C_VEL
LIN {X 0,Y 140.619,Z 619.128,A -85,B 0,C 180,E1 -24388.349,E2 -24388.349} C_VEL
LIN {X 0,Y 140.661,Z 619.021,A -85,B 0,C 180,E1 -24392.864,E2 -24392.864} C_VEL
LIN {X 0,Y 140.875,Z 618.435,A -85,B 0,C 180,E1 -24395.727,E2 -24395.727} C_VEL
LIN {X 0,Y 142.055,Z 616.106,A -85,B 0,C 180,E1 -24401.415,E2 -24401.415} C_VEL
LIN {X 0,Y 143.616,Z 613.233,A -85,B 0,C 180,E1 -24405.614,E2 -24405.614} C_VEL
LIN {X 0,Y 145.847,Z 609.335,A -85,B 0,C 180,E1 -24409.714,E2 -24409.714} C_VEL
LIN {X 0,Y 148.713,Z 604.305,A -85,B 0,C 180,E1 -24413.685,E2 -24413.685} C_VEL
LIN {X 0,Y 152.305,Z 597.966,A -85,B 0,C 180,E1 -24417.481,E2 -24417.481} C_VEL
LIN {X 0,Y 156.314,Z 590.069,A -85,B 0,C 180,E1 -24421.121,E2 -24421.121} C_VEL
LIN {X 0,Y 160.086,Z 581.958,A -85,B 0,C 180,E1 -24424.039,E2 -24424.039} C_VEL
LIN {X 0,Y 164.266,Z 572.093,A -85,B 0,C 180,E1 -24426.798,E2 -24426.798} C_VEL
LIN {X 0,Y 168.374,Z 560.977,A -85,B 0,C 180,E1 -24429.149,E2 -24429.149} C_VEL
LIN {X 0,Y 171.77,Z 550.078,A -85,B 0,C 180,E1 -24430.894,E2 -24430.894} C_VEL
LIN {X 0,Y 174.717,Z 538.027,A -85,B 0,C 180,E1 -24432.36,E2 -24432.36} C_VEL
LIN {X 0,Y 176.98,Z 525.47,A -85,B 0,C 180,E1 -24433.446,E2 -24433.446} C_VEL
LIN {X 0,Y 178.54,Z 512.484,A -85,B 0,C 180,E1 -24434.135,E2 -24434.135} C_VEL
LIN {X 0,Y 181.021,Z 474.93,A -85,B 0,C 180,E1 -24435.453,E2 -24435.453} C_VEL
LIN {X 0,Y 176.043,Z 462.981,A -85,B 0,C 180,E1 -24437.841,E2 -24437.841} C_VEL
LIN {X 0,Y 169.723,Z 452.039,A -85,B 0,C 180,E1 -24440.984,E2 -24440.984} C_VEL
LIN {X 0,Y 164.155,Z 443.59,A -85,B 0,C 180,E1 -24444.077,E2 -24444.077} C_VEL
LIN {X 0,Y 161.675,Z 440.014,A -85,B 0,C 180,E1 -24445.59,E2 -24445.59} C_VEL
LIN {X 0,Y 159.089,Z 436.447,A -85,B 0,C 180,E1 -24447.274,E2 -24447.274} C_VEL
LIN {X 0,Y 155.872,Z 432.153,A -85,B 0,C 180,E1 -24449.555,E2 -24449.555} C_VEL
LIN {X 0,Y 153.242,Z 428.996,A -85,B 0,C 180,E1 -24451.587,E2 -24451.587} C_VEL
LIN {X 0,Y 152.349,Z 427.466,A -85,B 0,C 180,E1 -24452.371,E2 -24452.371} C_VEL
LIN {X 0,Y 149.732,Z 425.164,A -85,B 0,C 180,E1 -24454.615,E2 -24454.615} C_VEL
LIN {X 0,Y 148.132,Z 422.219,A -85,B 0,C 180,E1 -24456.309,E2 -24456.309} C_VEL
LIN {X 0,Y 145.118,Z 419.965,A -85,B 0,C 180,E1 -24459.521,E2 -24459.521} C_VEL
LIN {X 0,Y 143.646,Z 417.511,A -85,B 0,C 180,E1 -24461.549,E2 -24461.549} C_VEL
LIN {X 0,Y 143.335,Z 416.121,A -85,B 0,C 180,E1 -24462.247,E2 -24462.247} C_VEL
LIN {X 0,Y 143.606,Z 416.092,A -85,B 0,C 180,E1 -24468.711,E2 -24468.711} C_VEL
LIN {X 0,Y 143.687,Z 416.071,A -85,B 0,C 180,E1 -24471.562,E2 -24471.562} C_VEL
LIN {X 0,Y 144.18,Z 416.008,A -85,B 0,C 180,E1 -24480,E2 -24480} C_VEL
LIN {X 0,Y 143.629,Z 416.094,A -85,B 0,C 180,E1 -24488.441,E2 -24488.441} C_VEL
LIN {X 0,Y 143.508,Z 416.091,A -85,B 0,C 180,E1 -24491.63,E2 -24491.63} C_VEL
LIN {X 0,Y 143.301,Z 416.119,A -85,B 0,C 180,E1 -24497.481,E2 -24497.481} C_VEL
LIN {X 0,Y 143.914,Z 418.258,A -85,B 0,C 180,E1 -24498.599,E2 -24498.599} C_VEL
LIN {X 0,Y 145.806,Z 420.721,A -85,B 0,C 180,E1 -24501.011,E2 -24501.011} C_VEL
LIN {X 0,Y 148.136,Z 422.251,A -85,B 0,C 180,E1 -24503.412,E2 -24503.412} C_VEL
LIN {X 0,Y 149.748,Z 425.213,A -85,B 0,C 180,E1 -24505.117,E2 -24505.117} C_VEL
LIN {X 0,Y 152.645,Z 427.913,A -85,B 0,C 180,E1 -24507.6,E2 -24507.6} C_VEL
LIN {X 0,Y 155.018,Z 431.35,A -85,B 0,C 180,E1 -24509.54,E2 -24509.54} C_VEL
LIN {X 0,Y 156.576,Z 433.037,A -85,B 0,C 180,E1 -24510.674,E2 -24510.674} C_VEL
LIN {X 0,Y 159.453,Z 436.865,A -85,B 0,C 180,E1 -24512.679,E2 -24512.679} C_VEL
LIN {X 0,Y 163.087,Z 442.359,A -85,B 0,C 180,E1 -24515.021,E2 -24515.021} C_VEL
LIN {X 0,Y 167.696,Z 450.448,A -85,B 0,C 180,E1 -24517.754,E2 -24517.754} C_VEL
LIN {X 0,Y 173.37,Z 461.939,A -85,B 0,C 180,E1 -24520.819,E2 -24520.819} C_VEL
LIN {X 0,Y 178.341,Z 473.802,A -85,B 0,C 180,E1 -24523.31,E2 -24523.31} C_VEL
LIN {X 0,Y 180.674,Z 480.195,A -85,B 0,C 180,E1 -24524.441,E2 -24524.441} C_VEL
LIN {X 0,Y 177.844,Z 521.74,A -85,B 0,C 180,E1 -24525.921,E2 -24525.921} C_VEL
LIN {X 0,Y 175.878,Z 535.545,A -85,B 0,C 180,E1 -24526.769,E2 -24526.769} C_VEL
LIN {X 0,Y 173.17,Z 548.324,A -85,B 0,C 180,E1 -24527.96,E2 -24527.96} C_VEL
LIN {X 0,Y 169.543,Z 560.979,A -85,B 0,C 180,E1 -24529.631,E2 -24529.631} C_VEL
LIN {X 0,Y 165.712,Z 572.24,A -85,B 0,C 180,E1 -24531.664,E2 -24531.664} C_VEL
LIN {X 0,Y 161.625,Z 582.382,A -85,B 0,C 180,E1 -24534.053,E2 -24534.053} C_VEL
LIN {X 0,Y 157.435,Z 591.522,A -85,B 0,C 180,E1 -24536.848,E2 -24536.848} C_VEL
LIN {X 0,Y 153.162,Z 600.254,A -85,B 0,C 180,E1 -24540.341,E2 -24540.341} C_VEL
LIN {X 0,Y 149.44,Z 607.613,A -85,B 0,C 180,E1 -24544.213,E2 -24544.213} C_VEL
LIN {X 0,Y 145.835,Z 614.05,A -85,B 0,C 180,E1 -24548.727,E2 -24548.727} C_VEL
LIN {X 0,Y 143.358,Z 618.47,A -85,B 0,C 180,E1 -24552.893,E2 -24552.893} C_VEL
LIN {X 0,Y 142.263,Z 620.765,A -85,B 0,C 180,E1 -24555.699,E2 -24555.699} C_VEL
LIN {X 0,Y 141.032,Z 623.474,A -85,B 0,C 180,E1 -24560.275,E2 -24560.275} C_VEL
LIN {X 0,Y 140.045,Z 624.501,A -85,B 0,C 180,E1 -24562.616,E2 -24562.616} C_VEL
LIN {X 0,Y 138.316,Z 625.235,A -85,B 0,C 180,E1 -24564.939,E2 -24564.939} C_VEL
LIN {X 0,Y 134.558,Z 625.798,A -85,B 0,C 180,E1 -24569.723,E2 -24569.723} C_VEL
LIN {X 0,Y 133.395,Z 625.425,A -85,B 0,C 180,E1 -24573.099,E2 -24573.099} C_VEL
LIN {X 0,Y 133.828,Z 623.816,A -85,B 0,C 180,E1 -24579.064,E2 -24579.064} C_VEL
LIN {X 0,Y 134.453,Z 622.406,A -85,B 0,C 180,E1 -24582.068,E2 -24582.068} C_VEL
LIN {X 0,Y 135.928,Z 619.454,A -85,B 0,C 180,E1 -24586.521,E2 -24586.521} C_VEL
LIN {X 0,Y 138.202,Z 615.468,A -85,B 0,C 180,E1 -24590.853,E2 -24590.853} C_VEL
LIN {X 0,Y 141.791,Z 609.342,A -85,B 0,C 180,E1 -24595.702,E2 -24595.702} C_VEL
LIN {X 0,Y 144.87,Z 603.891,A -85,B 0,C 180,E1 -24599.02,E2 -24599.02} C_VEL
LIN {X 0,Y 149.109,Z 595.852,A -85,B 0,C 180,E1 -24602.822,E2 -24602.822} C_VEL
LIN {X 0,Y 153.234,Z 587.663,A -85,B 0,C 180,E1 -24605.786,E2 -24605.786} C_VEL
LIN {X 0,Y 157.764,Z 577.676,A -85,B 0,C 180,E1 -24608.584,E2 -24608.584} C_VEL
LIN {X 0,Y 162.193,Z 566.384,A -85,B 0,C 180,E1 -24610.948,E2 -24610.948} C_VEL
LIN {X 0,Y 165.785,Z 555.317,A -85,B 0,C 180,E1 -24612.709,E2 -24612.709} C_VEL
LIN {X 0,Y 169.042,Z 543.033,A -85,B 0,C 180,E1 -24614.138,E2 -24614.138} C_VEL
LIN {X 0,Y 171.56,Z 530.229,A -85,B 0,C 180,E1 -24615.148,E2 -24615.148} C_VEL
LIN {X 0,Y 173.114,Z 517.007,A -85,B 0,C 180,E1 -24615.834,E2 -24615.834} C_VEL
LIN {X 0,Y 175.458,Z 482.108,A -85,B 0,C 180,E1 -24617.083,E2 -24617.083} C_VEL
LIN {X 0,Y 170.763,Z 469.663,A -85,B 0,C 180,E1 -24619.575,E2 -24619.575} C_VEL
LIN {X 0,Y 165.462,Z 458.141,A -85,B 0,C 180,E1 -24622.561,E2 -24622.561} C_VEL
LIN {X 0,Y 160.443,Z 448.777,A -85,B 0,C 180,E1 -24625.669,E2 -24625.669} C_VEL
LIN {X 0,Y 158.515,Z 445.485,A -85,B 0,C 180,E1 -24626.962,E2 -24626.962} C_VEL
LIN {X 0,Y 155.896,Z 441.855,A -85,B 0,C 180,E1 -24628.774,E2 -24628.774} C_VEL
LIN {X 0,Y 153.383,Z 438.27,A -85,B 0,C 180,E1 -24630.679,E2 -24630.679} C_VEL
LIN {X 0,Y 150.63,Z 434.683,A -85,B 0,C 180,E1 -24632.949,E2 -24632.949} C_VEL
LIN {X 0,Y 149.783,Z 433.635,A -85,B 0,C 180,E1 -24633.695,E2 -24633.695} C_VEL
LIN {X 0,Y 146.986,Z 430.463,A -85,B 0,C 180,E1 -24636.347,E2 -24636.347} C_VEL
LIN {X 0,Y 146.1,Z 428.682,A -85,B 0,C 180,E1 -24637.367,E2 -24637.367} C_VEL
LIN {X 0,Y 143.332,Z 426.419,A -85,B 0,C 180,E1 -24640.486,E2 -24640.486} C_VEL
LIN {X 0,Y 141.737,Z 423.354,A -85,B 0,C 180,E1 -24642.878,E2 -24642.878} C_VEL
LIN {X 0,Y 141.397,Z 422.954,A -85,B 0,C 180,E1 -24643.394,E2 -24643.394} C_VEL
LIN {X 0,Y 138.556,Z 421.208,A -85,B 0,C 180,E1 -24648.294,E2 -24648.294} C_VEL
LIN {X 0,Y 136.642,Z 417.415,A -85,B 0,C 180,E1 -24654.836,E2 -24654.836} C_VEL
LIN {X 0,Y 136.614,Z 416.954,A -85,B 0,C 180,E1 -24655.574,E2 -24655.574} C_VEL
LIN {X 0,Y 137.134,Z 416.891,A -85,B 0,C 180,E1 -24660,E2 -24660} C_VEL
LIN {X 0,Y 136.631,Z 417.166,A -85,B 0,C 180,E1 -24665.35,E2 -24665.35} C_VEL
LIN {X 0,Y 137.929,Z 420.368,A -85,B 0,C 180,E1 -24670.541,E2 -24670.541} C_VEL
LIN {X 0,Y 140.459,Z 422.62,A -85,B 0,C 180,E1 -24675.602,E2 -24675.602} C_VEL
LIN {X 0,Y 141.696,Z 423.119,A -85,B 0,C 180,E1 -24677.406,E2 -24677.406} C_VEL
LIN {X 0,Y 142.95,Z 425.902,A -85,B 0,C 180,E1 -24679.382,E2 -24679.382} C_VEL
LIN {X 0,Y 145.459,Z 428.344,A -85,B 0,C 180,E1 -24682.359,E2 -24682.359} C_VEL
LIN {X 0,Y 146.235,Z 428.978,A -85,B 0,C 180,E1 -24683.172,E2 -24683.172} C_VEL
LIN {X 0,Y 148.443,Z 432.41,A -85,B 0,C 180,E1 -24685.488,E2 -24685.488} C_VEL
LIN {X 0,Y 150.462,Z 434.336,A -85,B 0,C 180,E1 -24687.267,E2 -24687.267} C_VEL
LIN {X 0,Y 153.113,Z 438.033,A -85,B 0,C 180,E1 -24689.496,E2 -24689.496} C_VEL
LIN {X 0,Y 154.387,Z 439.674,A -85,B 0,C 180,E1 -24690.476,E2 -24690.476} C_VEL
LIN {X 0,Y 157.762,Z 444.381,A -85,B 0,C 180,E1 -24692.904,E2 -24692.904} C_VEL
LIN {X 0,Y 162.349,Z 451.144,A -85,B 0,C 180,E1 -24695.849,E2 -24695.849} C_VEL
LIN {X 0,Y 168.574,Z 461.389,A -85,B 0,C 180,E1 -24699.382,E2 -24699.382} C_VEL
LIN {X 0,Y 172.584,Z 468.947,A -85,B 0,C 180,E1 -24701.457,E2 -24701.457} C_VEL
LIN {X 0,Y 175.791,Z 477.057,A -85,B 0,C 180,E1 -24703.113,E2 -24703.113} C_VEL
LIN {X 0,Y 173.762,Z 506.529,A -85,B 0,C 180,E1 -24704.136,E2 -24704.136} C_VEL
LIN {X 0,Y 172.433,Z 521.058,A -85,B 0,C 180,E1 -24704.796,E2 -24704.796} C_VEL
LIN {X 0,Y 170.093,Z 534.472,A -85,B 0,C 180,E1 -24705.793,E2 -24705.793} C_VEL
LIN {X 0,Y 167.508,Z 545.631,A -85,B 0,C 180,E1 -24707.017,E2 -24707.017} C_VEL
LIN {X 0,Y 164.027,Z 557.578,A -85,B 0,C 180,E1 -24708.795,E2 -24708.795} C_VEL
LIN {X 0,Y 160.159,Z 568.225,A -85,B 0,C 180,E1 -24710.892,E2 -24710.892} C_VEL
LIN {X 0,Y 156.08,Z 577.931,A -85,B 0,C 180,E1 -24713.372,E2 -24713.372} C_VEL
LIN {X 0,Y 151.929,Z 586.761,A -85,B 0,C 180,E1 -24716.283,E2 -24716.283} C_VEL
LIN {X 0,Y 147.527,Z 595.369,A -85,B 0,C 180,E1 -24719.987,E2 -24719.987} C_VEL
LIN {X 0,Y 143.504,Z 602.237,A -85,B 0,C 180,E1 -24723.848,E2 -24723.848} C_VEL
LIN {X 0,Y 140.172,Z 607.733,A -85,B 0,C 180,E1 -24727.912,E2 -24727.912} C_VEL
LIN {X 0,Y 137.529,Z 612.044,A -85,B 0,C 180,E1 -24732.145,E2 -24732.145} C_VEL
LIN {X 0,Y 136.157,Z 614.324,A -85,B 0,C 180,E1 -24735.044,E2 -24735.044} C_VEL
LIN {X 0,Y 135.101,Z 616.175,A -85,B 0,C 180,E1 -24737.991,E2 -24737.991} C_VEL
LIN {X 0,Y 134.304,Z 617.565,A -85,B 0,C 180,E1 -24740.968,E2 -24740.968} C_VEL
LIN {X 0,Y 133.575,Z 619.158,A -85,B 0,C 180,E1 -24746.985,E2 -24746.985} C_VEL
LIN {X 0,Y 133.533,Z 619.383,A -85,B 0,C 180,E1 -24750.001,E2 -24750.001} C_VEL
LIN {X 0,Y 133.575,Z 619.188,A -85,B 0,C 180,E1 -24753.017,E2 -24753.017} C_VEL
LIN {X 0,Y 134.305,Z 617.633,A -85,B 0,C 180,E1 -24759.033,E2 -24759.033} C_VEL
LIN {X 0,Y 135.102,Z 616.272,A -85,B 0,C 180,E1 -24762.011,E2 -24762.011} C_VEL
LIN {X 0,Y 136.774,Z 613.4,A -85,B 0,C 180,E1 -24766.417,E2 -24766.417} C_VEL
LIN {X 0,Y 139.158,Z 609.501,A -85,B 0,C 180,E1 -24770.704,E2 -24770.704} C_VEL
LIN {X 0,Y 142.238,Z 604.471,A -85,B 0,C 180,E1 -24774.834,E2 -24774.834} C_VEL
LIN {X 0,Y 146.035,Z 598.131,A -85,B 0,C 180,E1 -24778.768,E2 -24778.768} C_VEL
LIN {X 0,Y 150.024,Z 590.733,A -85,B 0,C 180,E1 -24782.314,E2 -24782.314} C_VEL
LIN {X 0,Y 154.239,Z 582.123,A -85,B 0,C 180,E1 -24785.519,E2 -24785.519} C_VEL
LIN {X 0,Y 158.633,Z 572.257,A -85,B 0,C 180,E1 -24788.335,E2 -24788.335} C_VEL
LIN {X 0,Y 162.948,Z 561.139,A -85,B 0,C 180,E1 -24790.72,E2 -24790.72} C_VEL
LIN {X 0,Y 166.468,Z 550.239,A -85,B 0,C 180,E1 -24792.493,E2 -24792.493} C_VEL
LIN {X 0,Y 169.546,Z 538.187,A -85,B 0,C 180,E1 -24793.974,E2 -24793.974} C_VEL
LIN {X 0,Y 171.952,Z 525.301,A -85,B 0,C 180,E1 -24795.091,E2 -24795.091} C_VEL
LIN {X 0,Y 173.615,Z 511.492,A -85,B 0,C 180,E1 -24795.813,E2 -24795.813} C_VEL
LIN {X 0,Y 175.95,Z 477.067,A -85,B 0,C 180,E1 -24797.039,E2 -24797.039} C_VEL
LIN {X 0,Y 171.746,Z 467.026,A -85,B 0,C 180,E1 -24799.202,E2 -24799.202} C_VEL
LIN {X 0,Y 165.85,Z 456.609,A -85,B 0,C 180,E1 -24802.355,E2 -24802.355} C_VEL
LIN {X 0,Y 160.997,Z 449.043,A -85,B 0,C 180,E1 -24805.245,E2 -24805.245} C_VEL
LIN {X 0,Y 156.728,Z 442.735,A -85,B 0,C 180,E1 -24808.11,E2 -24808.11} C_VEL
LIN {X 0,Y 153.369,Z 438.249,A -85,B 0,C 180,E1 -24810.618,E2 -24810.618} C_VEL
LIN {X 0,Y 150.535,Z 434.409,A -85,B 0,C 180,E1 -24813.002,E2 -24813.002} C_VEL
LIN {X 0,Y 147.102,Z 430.595,A -85,B 0,C 180,E1 -24816.227,E2 -24816.227} C_VEL
LIN {X 0,Y 146.116,Z 428.667,A -85,B 0,C 180,E1 -24817.369,E2 -24817.369} C_VEL
LIN {X 0,Y 143.517,Z 426.597,A -85,B 0,C 180,E1 -24820.326,E2 -24820.326} C_VEL
LIN {X 0,Y 141.911,Z 423.768,A -85,B 0,C 180,E1 -24822.714,E2 -24822.714} C_VEL
LIN {X 0,Y 141.62,Z 422.994,A -85,B 0,C 180,E1 -24823.235,E2 -24823.235} C_VEL
LIN {X 0,Y 138.927,Z 421.504,A -85,B 0,C 180,E1 -24827.843,E2 -24827.843} C_VEL
LIN {X 0,Y 136.726,Z 417.488,A -85,B 0,C 180,E1 -24835.762,E2 -24835.762} C_VEL
LIN {X 0,Y 136.735,Z 416.948,A -85,B 0,C 180,E1 -24836.685,E2 -24836.685} C_VEL
LIN {X 0,Y 137.137,Z 416.884,A -85,B 0,C 180,E1 -24840,E2 -24840} C_VEL
LIN {X 0,Y 136.713,Z 417.121,A -85,B 0,C 180,E1 -24843.592,E2 -24843.592} C_VEL
LIN {X 0,Y 137.313,Z 419.425,A -85,B 0,C 180,E1 -24847.351,E2 -24847.351} C_VEL
LIN {X 0,Y 140.316,Z 422.55,A -85,B 0,C 180,E1 -24854.503,E2 -24854.503} C_VEL
LIN {X 0,Y 141.665,Z 423.189,A -85,B 0,C 180,E1 -24856.574,E2 -24856.574} C_VEL
LIN {X 0,Y 143.197,Z 426.273,A -85,B 0,C 180,E1 -24858.975,E2 -24858.975} C_VEL
LIN {X 0,Y 145.844,Z 428.537,A -85,B 0,C 180,E1 -24862.07,E2 -24862.07} C_VEL
LIN {X 0,Y 146.322,Z 429.129,A -85,B 0,C 180,E1 -24862.597,E2 -24862.597} C_VEL
LIN {X 0,Y 148.28,Z 432.198,A -85,B 0,C 180,E1 -24864.688,E2 -24864.688} C_VEL
LIN {X 0,Y 150.513,Z 434.428,A -85,B 0,C 180,E1 -24866.698,E2 -24866.698} C_VEL
LIN {X 0,Y 153.411,Z 438.288,A -85,B 0,C 180,E1 -24869.127,E2 -24869.127} C_VEL
LIN {X 0,Y 157.739,Z 444.272,A -85,B 0,C 180,E1 -24872.321,E2 -24872.321} C_VEL
LIN {X 0,Y 160.118,Z 448.082,A -85,B 0,C 180,E1 -24873.935,E2 -24873.935} C_VEL
LIN {X 0,Y 164.204,Z 455.531,A -85,B 0,C 180,E1 -24876.526,E2 -24876.526} C_VEL
LIN {X 0,Y 169.479,Z 466.545,A -85,B 0,C 180,E1 -24879.58,E2 -24879.58} C_VEL
LIN {X 0,Y 174.32,Z 478.598,A -85,B 0,C 180,E1 -24882.185,E2 -24882.185} C_VEL
LIN {X 0,Y 175.614,Z 482.389,A -85,B 0,C 180,E1 -24882.87,E2 -24882.87} C_VEL
LIN {X 0,Y 172.844,Z 521.243,A -85,B 0,C 180,E1 -24884.262,E2 -24884.262} C_VEL
LIN {X 0,Y 170.892,Z 534.858,A -85,B 0,C 180,E1 -24885.104,E2 -24885.104} C_VEL
LIN {X 0,Y 168.237,Z 547.061,A -85,B 0,C 180,E1 -24886.219,E2 -24886.219} C_VEL
LIN {X 0,Y 164.746,Z 559.234,A -85,B 0,C 180,E1 -24887.786,E2 -24887.786} C_VEL
LIN {X 0,Y 160.659,Z 570.782,A -85,B 0,C 180,E1 -24889.816,E2 -24889.816} C_VEL
LIN {X 0,Y 156.395,Z 581.186,A -85,B 0,C 180,E1 -24892.245,E2 -24892.245} C_VEL
LIN {X 0,Y 152.377,Z 589.691,A -85,B 0,C 180,E1 -24894.792,E2 -24894.792} C_VEL
LIN {X 0,Y 148.361,Z 597.54,A -85,B 0,C 180,E1 -24897.796,E2 -24897.796} C_VEL
LIN {X 0,Y 144.334,Z 605.213,A -85,B 0,C 180,E1 -24901.656,E2 -24901.656} C_VEL
LIN {X 0,Y 140.181,Z 612.29,A -85,B 0,C 180,E1 -24906.353,E2 -24906.353} C_VEL
LIN {X 0,Y 137.332,Z 616.997,A -85,B 0,C 180,E1 -24910.57,E2 -24910.57} C_VEL
LIN {X 0,Y 135.373,Z 620.598,A -85,B 0,C 180,E1 -24914.954,E2 -24914.954} C_VEL
LIN {X 0,Y 133.973,Z 623.442,A -85,B 0,C 180,E1 -24920.054,E2 -24920.054} C_VEL
LIN {X 0,Y 133.467,Z 624.847,A -85,B 0,C 180,E1 -24923.954,E2 -24923.954} C_VEL
LIN {X 0,Y 133.397,Z 625.457,A -85,B 0,C 180,E1 -24926.979,E2 -24926.979} C_VEL
LIN {X 0,Y 133.474,Z 625.67,A -85,B 0,C 180,E1 -24929.999,E2 -24929.999} C_VEL
LIN {X 0,Y 133.395,Z 625.425,A -85,B 0,C 180,E1 -24933.099,E2 -24933.099} C_VEL
LIN {X 0,Y 132.756,Z 624.938,A -85,B 0,C 180,E1 -24935.613,E2 -24935.613} C_VEL
LIN {X 0,Y 130.39,Z 623.565,A -85,B 0,C 180,E1 -24939.763,E2 -24939.763} C_VEL
LIN {X 0,Y 128.755,Z 621.979,A -85,B 0,C 180,E1 -24943.145,E2 -24943.145} C_VEL
LIN {X 0,Y 128.528,Z 620.471,A -85,B 0,C 180,E1 -24945.704,E2 -24945.704} C_VEL
LIN {X 0,Y 128.754,Z 619.895,A -85,B 0,C 180,E1 -24946.544,E2 -24946.544} C_VEL
LIN {X 0,Y 131.565,Z 615.299,A -85,B 0,C 180,E1 -24951.958,E2 -24951.958} C_VEL
LIN {X 0,Y 135.421,Z 609.173,A -85,B 0,C 180,E1 -24957.007,E2 -24957.007} C_VEL
LIN {X 0,Y 138.703,Z 603.596,A -85,B 0,C 180,E1 -24960.528,E2 -24960.528} C_VEL
LIN {X 0,Y 143.162,Z 595.681,A -85,B 0,C 180,E1 -24964.371,E2 -24964.371} C_VEL
LIN {X 0,Y 147.508,Z 587.492,A -85,B 0,C 180,E1 -24967.407,E2 -24967.407} C_VEL
LIN {X 0,Y 152.264,Z 577.505,A -85,B 0,C 180,E1 -24970.255,E2 -24970.255} C_VEL
LIN {X 0,Y 156.905,Z 566.213,A -85,B 0,C 180,E1 -24972.646,E2 -24972.646} C_VEL
LIN {X 0,Y 160.64,Z 555.145,A -85,B 0,C 180,E1 -24974.427,E2 -24974.427} C_VEL
LIN {X 0,Y 164.025,Z 542.859,A -85,B 0,C 180,E1 -24975.864,E2 -24975.864} C_VEL
LIN {X 0,Y 166.623,Z 530.035,A -85,B 0,C 180,E1 -24976.883,E2 -24976.883} C_VEL
LIN {X 0,Y 168.269,Z 516.698,A -85,B 0,C 180,E1 -24977.568,E2 -24977.568} C_VEL
LIN {X 0,Y 170.469,Z 484.044,A -85,B 0,C 180,E1 -24978.785,E2 -24978.785} C_VEL
LIN {X 0,Y 165.987,Z 472.136,A -85,B 0,C 180,E1 -24981.37,E2 -24981.37} C_VEL
LIN {X 0,Y 160.993,Z 461.211,A -85,B 0,C 180,E1 -24984.445,E2 -24984.445} C_VEL
LIN {X 0,Y 156.231,Z 452.024,A -85,B 0,C 180,E1 -24987.711,E2 -24987.711} C_VEL
LIN {X 0,Y 153.348,Z 447.851,A -85,B 0,C 180,E1 -24989.821,E2 -24989.821} C_VEL
LIN {X 0,Y 150.83,Z 444.219,A -85,B 0,C 180,E1 -24991.85,E2 -24991.85} C_VEL
LIN {X 0,Y 147.706,Z 440.028,A -85,B 0,C 180,E1 -24994.645,E2 -24994.645} C_VEL
LIN {X 0,Y 144.824,Z 436.43,A -85,B 0,C 180,E1 -24997.597,E2 -24997.597} C_VEL
LIN {X 0,Y 144.11,Z 435.213,A -85,B 0,C 180,E1 -24998.449,E2 -24998.449} C_VEL
LIN {X 0,Y 141.434,Z 432.567,A -85,B 0,C 180,E1 -25001.766,E2 -25001.766} C_VEL
LIN {X 0,Y 140.082,Z 429.884,A -85,B 0,C 180,E1 -25003.982,E2 -25003.982} C_VEL
LIN {X 0,Y 137.341,Z 427.984,A -85,B 0,C 180,E1 -25009.039,E2 -25009.039} C_VEL
LIN {X 0,Y 135.654,Z 424.242,A -85,B 0,C 180,E1 -25015.543,E2 -25015.543} C_VEL
LIN {X 0,Y 135.453,Z 423.924,A -85,B 0,C 180,E1 -25017.026,E2 -25017.026} C_VEL
LIN {X 0,Y 135.408,Z 423.916,A -85,B 0,C 180,E1 -25022.975,E2 -25022.975} C_VEL
LIN {X 0,Y 135.659,Z 424.191,A -85,B 0,C 180,E1 -25024.829,E2 -25024.829} C_VEL
LIN {X 0,Y 137.859,Z 428.531,A -85,B 0,C 180,E1 -25032.513,E2 -25032.513} C_VEL
LIN {X 0,Y 140.236,Z 430.133,A -85,B 0,C 180,E1 -25036.655,E2 -25036.655} C_VEL
LIN {X 0,Y 141.891,Z 433.177,A -85,B 0,C 180,E1 -25039.25,E2 -25039.25} C_VEL
LIN {X 0,Y 144.45,Z 435.661,A -85,B 0,C 180,E1 -25042.321,E2 -25042.321} C_VEL
LIN {X 0,Y 146.7,Z 439.049,A -85,B 0,C 180,E1 -25044.784,E2 -25044.784} C_VEL
LIN {X 0,Y 148.45,Z 440.949,A -85,B 0,C 180,E1 -25046.424,E2 -25046.424} C_VEL
LIN {X 0,Y 152.029,Z 445.912,A -85,B 0,C 180,E1 -25049.513,E2 -25049.513} C_VEL
LIN {X 0,Y 155.327,Z 450.691,A -85,B 0,C 180,E1 -25052.023,E2 -25052.023} C_VEL
LIN {X 0,Y 159.381,Z 456.899,A -85,B 0,C 180,E1 -25054.784,E2 -25054.784} C_VEL
LIN {X 0,Y 165.178,Z 466.753,A -85,B 0,C 180,E1 -25058.286,E2 -25058.286} C_VEL
LIN {X 0,Y 168.796,Z 473.897,A -85,B 0,C 180,E1 -25060.291,E2 -25060.291} C_VEL
LIN {X 0,Y 170.868,Z 479.241,A -85,B 0,C 180,E1 -25061.443,E2 -25061.443} C_VEL
LIN {X 0,Y 168.96,Z 506.082,A -85,B 0,C 180,E1 -25062.392,E2 -25062.392} C_VEL
LIN {X 0,Y 167.617,Z 520.509,A -85,B 0,C 180,E1 -25063.034,E2 -25063.034} C_VEL
LIN {X 0,Y 165.35,Z 533.349,A -85,B 0,C 180,E1 -25063.953,E2 -25063.953} C_VEL
LIN {X 0,Y 162.385,Z 545.805,A -85,B 0,C 180,E1 -25065.308,E2 -25065.308} C_VEL
LIN {X 0,Y 158.77,Z 557.75,A -85,B 0,C 180,E1 -25067.111,E2 -25067.111} C_VEL
LIN {X 0,Y 154.714,Z 568.396,A -85,B 0,C 180,E1 -25069.232,E2 -25069.232} C_VEL
LIN {X 0,Y 150.438,Z 578.101,A -85,B 0,C 180,E1 -25071.757,E2 -25071.757} C_VEL
LIN {X 0,Y 146.063,Z 586.931,A -85,B 0,C 180,E1 -25074.733,E2 -25074.733} C_VEL
LIN {X 0,Y 141.415,Z 595.538,A -85,B 0,C 180,E1 -25078.546,E2 -25078.546} C_VEL
LIN {X 0,Y 137.168,Z 602.406,A -85,B 0,C 180,E1 -25082.541,E2 -25082.541} C_VEL
LIN {X 0,Y 133.595,Z 607.902,A -85,B 0,C 180,E1 -25086.762,E2 -25086.762} C_VEL
LIN {X 0,Y 130.772,Z 612.213,A -85,B 0,C 180,E1 -25091.189,E2 -25091.189} C_VEL
LIN {X 0,Y 129.308,Z 614.492,A -85,B 0,C 180,E1 -25094.232,E2 -25094.232} C_VEL
LIN {X 0,Y 128.175,Z 616.343,A -85,B 0,C 180,E1 -25097.331,E2 -25097.331} C_VEL
LIN {X 0,Y 126.753,Z 618.72,A -85,B 0,C 180,E1 -25103.634,E2 -25103.634} C_VEL
LIN {X 0,Y 126.502,Z 619.325,A -85,B 0,C 180,E1 -25106.816,E2 -25106.816} C_VEL
LIN {X 0,Y 126.447,Z 619.55,A -85,B 0,C 180,E1 -25110.001,E2 -25110.001} C_VEL
LIN {X 0,Y 126.502,Z 619.354,A -85,B 0,C 180,E1 -25113.185,E2 -25113.185} C_VEL
LIN {X 0,Y 127.286,Z 617.8,A -85,B 0,C 180,E1 -25119.535,E2 -25119.535} C_VEL
LIN {X 0,Y 128.175,Z 616.439,A -85,B 0,C 180,E1 -25122.67,E2 -25122.67} C_VEL
LIN {X 0,Y 129.966,Z 613.566,A -85,B 0,C 180,E1 -25127.303,E2 -25127.303} C_VEL
LIN {X 0,Y 132.515,Z 609.668,A -85,B 0,C 180,E1 -25131.793,E2 -25131.793} C_VEL
LIN {X 0,Y 135.831,Z 604.636,A -85,B 0,C 180,E1 -25136.092,E2 -25136.092} C_VEL
LIN {X 0,Y 139.844,Z 598.296,A -85,B 0,C 180,E1 -25140.17,E2 -25140.17} C_VEL
LIN {X 0,Y 143.805,Z 591.395,A -85,B 0,C 180,E1 -25143.612,E2 -25143.612} C_VEL
LIN {X 0,Y 148.516,Z 582.287,A -85,B 0,C 180,E1 -25147.111,E2 -25147.111} C_VEL
LIN {X 0,Y 153.138,Z 572.42,A -85,B 0,C 180,E1 -25149.98,E2 -25149.98} C_VEL
LIN {X 0,Y 157.64,Z 561.301,A -85,B 0,C 180,E1 -25152.402,E2 -25152.402} C_VEL
LIN {X 0,Y 161.303,Z 550.401,A -85,B 0,C 180,E1 -25154.198,E2 -25154.198} C_VEL
LIN {X 0,Y 164.528,Z 538.346,A -85,B 0,C 180,E1 -25155.685,E2 -25155.685} C_VEL
LIN {X 0,Y 167.05,Z 525.314,A -85,B 0,C 180,E1 -25156.821,E2 -25156.821} C_VEL
LIN {X 0,Y 168.71,Z 512.067,A -85,B 0,C 180,E1 -25157.523,E2 -25157.523} C_VEL
LIN {X 0,Y 171.06,Z 479.486,A -85,B 0,C 180,E1 -25158.686,E2 -25158.686} C_VEL
LIN {X 0,Y 167.733,Z 471.389,A -85,B 0,C 180,E1 -25160.536,E2 -25160.536} C_VEL
LIN {X 0,Y 162.411,Z 461.771,A -85,B 0,C 180,E1 -25163.586,E2 -25163.586} C_VEL
LIN {X 0,Y 156.85,Z 452.677,A -85,B 0,C 180,E1 -25167.202,E2 -25167.202} C_VEL
LIN {X 0,Y 153.376,Z 447.772,A -85,B 0,C 180,E1 -25169.732,E2 -25169.732} C_VEL
LIN {X 0,Y 150.789,Z 444.146,A -85,B 0,C 180,E1 -25171.829,E2 -25171.829} C_VEL
LIN {X 0,Y 147.812,Z 440.073,A -85,B 0,C 180,E1 -25174.53,E2 -25174.53} C_VEL
LIN {X 0,Y 145.11,Z 436.847,A -85,B 0,C 180,E1 -25177.291,E2 -25177.291} C_VEL
LIN {X 0,Y 144.143,Z 435.204,A -85,B 0,C 180,E1 -25178.454,E2 -25178.454} C_VEL
LIN {X 0,Y 141.419,Z 432.502,A -85,B 0,C 180,E1 -25181.904,E2 -25181.904} C_VEL
LIN {X 0,Y 140.191,Z 429.91,A -85,B 0,C 180,E1 -25183.995,E2 -25183.995} C_VEL
LIN {X 0,Y 137.601,Z 428.162,A -85,B 0,C 180,E1 -25188.843,E2 -25188.843} C_VEL
LIN {X 0,Y 135.775,Z 424.316,A -85,B 0,C 180,E1 -25196.476,E2 -25196.476} C_VEL
LIN {X 0,Y 135.747,Z 423.966,A -85,B 0,C 180,E1 -25197.032,E2 -25197.032} C_VEL
LIN {X 0,Y 135.645,Z 423.895,A -85,B 0,C 180,E1 -25201.484,E2 -25201.484} C_VEL
LIN {X 0,Y 135.783,Z 424.373,A -85,B 0,C 180,E1 -25203.338,E2 -25203.338} C_VEL
LIN {X 0,Y 137.384,Z 427.987,A -85,B 0,C 180,E1 -25210.347,E2 -25210.347} C_VEL
LIN {X 0,Y 140.23,Z 430.12,A -85,B 0,C 180,E1 -25215.814,E2 -25215.814} C_VEL
LIN {X 0,Y 142.078,Z 433.441,A -85,B 0,C 180,E1 -25218.755,E2 -25218.755} C_VEL
LIN {X 0,Y 144.493,Z 435.707,A -85,B 0,C 180,E1 -25221.677,E2 -25221.677} C_VEL
LIN {X 0,Y 146.78,Z 439.081,A -85,B 0,C 180,E1 -25224.204,E2 -25224.204} C_VEL
LIN {X 0,Y 148.493,Z 440.968,A -85,B 0,C 180,E1 -25225.831,E2 -25225.831} C_VEL
LIN {X 0,Y 152.15,Z 446.04,A -85,B 0,C 180,E1 -25229.013,E2 -25229.013} C_VEL
LIN {X 0,Y 155.227,Z 450.498,A -85,B 0,C 180,E1 -25231.377,E2 -25231.377} C_VEL
LIN {X 0,Y 157.342,Z 454.02,A -85,B 0,C 180,E1 -25232.901,E2 -25232.901} C_VEL
LIN {X 0,Y 161.167,Z 461.428,A -85,B 0,C 180,E1 -25235.495,E2 -25235.495} C_VEL
LIN {X 0,Y 166.127,Z 472.261,A -85,B 0,C 180,E1 -25238.556,E2 -25238.556} C_VEL
LIN {X 0,Y 170.457,Z 483.759,A -85,B 0,C 180,E1 -25241.064,E2 -25241.064} C_VEL
LIN {X 0,Y 170.702,Z 484.502,A -85,B 0,C 180,E1 -25241.204,E2 -25241.204} C_VEL
LIN {X 0,Y 167.969,Z 521.105,A -85,B 0,C 180,E1 -25242.53,E2 -25242.53} C_VEL
LIN {X 0,Y 166.014,Z 534.301,A -85,B 0,C 180,E1 -25243.343,E2 -25243.343} C_VEL
LIN {X 0,Y 163.173,Z 546.9,A -85,B 0,C 180,E1 -25244.49,E2 -25244.49} C_VEL
LIN {X 0,Y 159.572,Z 559.072,A -85,B 0,C 180,E1 -25246.077,E2 -25246.077} C_VEL
LIN {X 0,Y 155.301,Z 570.619,A -85,B 0,C 180,E1 -25248.125,E2 -25248.125} C_VEL
LIN {X 0,Y 150.832,Z 581.022,A -85,B 0,C 180,E1 -25250.59,E2 -25250.59} C_VEL
LIN {X 0,Y 146.63,Z 589.526,A -85,B 0,C 180,E1 -25253.192,E2 -25253.192} C_VEL
LIN {X 0,Y 141.584,Z 598.746,A -85,B 0,C 180,E1 -25256.905,E2 -25256.905} C_VEL
LIN {X 0,Y 137.431,Z 606.173,A -85,B 0,C 180,E1 -25260.937,E2 -25260.937} C_VEL
LIN {X 0,Y 133.66,Z 612.123,A -85,B 0,C 180,E1 -25265.124,E2 -25265.124} C_VEL
LIN {X 0,Y 130.634,Z 616.83,A -85,B 0,C 180,E1 -25269.531,E2 -25269.531} C_VEL
LIN {X 0,Y 128.51,Z 620.431,A -85,B 0,C 180,E1 -25274.13,E2 -25274.13} C_VEL
LIN {X 0,Y 127.484,Z 622.288,A -85,B 0,C 180,E1 -25277.26,E2 -25277.26} C_VEL
LIN {X 0,Y 126.798,Z 623.683,A -85,B 0,C 180,E1 -25280.428,E2 -25280.428} C_VEL
LIN {X 0,Y 126.41,Z 624.68,A -85,B 0,C 180,E1 -25283.615,E2 -25283.615} C_VEL
LIN {X 0,Y 126.303,Z 625.29,A -85,B 0,C 180,E1 -25286.81,E2 -25286.81} C_VEL
LIN {X 0,Y 126.389,Z 625.503,A -85,B 0,C 180,E1 -25289.999,E2 -25289.999} C_VEL
LIN {X 0,Y 126.303,Z 625.274,A -85,B 0,C 180,E1 -25293.189,E2 -25293.189} C_VEL
LIN {X 0,Y 126.412,Z 624.655,A -85,B 0,C 180,E1 -25296.383,E2 -25296.383} C_VEL
LIN {X 0,Y 126.797,Z 623.648,A -85,B 0,C 180,E1 -25299.571,E2 -25299.571} C_VEL
LIN {X 0,Y 127.483,Z 622.237,A -85,B 0,C 180,E1 -25302.739,E2 -25302.739} C_VEL
LIN {X 0,Y 128.754,Z 619.895,A -85,B 0,C 180,E1 -25306.544,E2 -25306.544} C_VEL
LIN {X 0,Y 129.184,Z 618.083,A -85,B 0,C 180,E1 -25309.037,E2 -25309.037} C_VEL
LIN {X 0,Y 128.715,Z 614.659,A -85,B 0,C 180,E1 -25313.168,E2 -25313.168} C_VEL
LIN {X 0,Y 128.807,Z 610.541,A -85,B 0,C 180,E1 -25317.18,E2 -25317.18} C_VEL
LIN {X 0,Y 130.069,Z 607.641,A -85,B 0,C 180,E1 -25319.389,E2 -25319.389} C_VEL
LIN {X 0,Y 134.053,Z 601.078,A -85,B 0,C 180,E1 -25323.4,E2 -25323.4} C_VEL
LIN {X 0,Y 139.115,Z 592.427,A -85,B 0,C 180,E1 -25327.317,E2 -25327.317} C_VEL
LIN {X 0,Y 143.875,Z 583.564,A -85,B 0,C 180,E1 -25330.333,E2 -25330.333} C_VEL
LIN {X 0,Y 148.512,Z 573.836,A -85,B 0,C 180,E1 -25332.864,E2 -25332.864} C_VEL
LIN {X 0,Y 152.852,Z 563.182,A -85,B 0,C 180,E1 -25334.985,E2 -25334.985} C_VEL
LIN {X 0,Y 156.799,Z 551.25,A -85,B 0,C 180,E1 -25336.748,E2 -25336.748} C_VEL
LIN {X 0,Y 160.064,Z 538.828,A -85,B 0,C 180,E1 -25338.046,E2 -25338.046} C_VEL
LIN {X 0,Y 162.446,Z 526.293,A -85,B 0,C 180,E1 -25338.937,E2 -25338.937} C_VEL
LIN {X 0,Y 163.969,Z 511.314,A -85,B 0,C 180,E1 -25339.599,E2 -25339.599} C_VEL
LIN {X 0,Y 165.762,Z 486.415,A -85,B 0,C 180,E1 -25340.508,E2 -25340.508} C_VEL
LIN {X 0,Y 161.542,Z 475.066,A -85,B 0,C 180,E1 -25343.161,E2 -25343.161} C_VEL
LIN {X 0,Y 157.088,Z 465.045,A -85,B 0,C 180,E1 -25346.166,E2 -25346.166} C_VEL
LIN {X 0,Y 152.939,Z 457,A -85,B 0,C 180,E1 -25349.255,E2 -25349.255} C_VEL
LIN {X 0,Y 148.701,Z 450.574,A -85,B 0,C 180,E1 -25352.751,E2 -25352.751} C_VEL
LIN {X 0,Y 145.528,Z 446.255,A -85,B 0,C 180,E1 -25355.764,E2 -25355.764} C_VEL
LIN {X 0,Y 142.783,Z 442.499,A -85,B 0,C 180,E1 -25358.819,E2 -25358.819} C_VEL
LIN {X 0,Y 142.036,Z 441.559,A -85,B 0,C 180,E1 -25359.735,E2 -25359.735} C_VEL
LIN {X 0,Y 139.484,Z 438.466,A -85,B 0,C 180,E1 -25363.29,E2 -25363.29} C_VEL
LIN {X 0,Y 138.564,Z 436.672,A -85,B 0,C 180,E1 -25364.934,E2 -25364.934} C_VEL
LIN {X 0,Y 135.96,Z 434.525,A -85,B 0,C 180,E1 -25370.312,E2 -25370.312} C_VEL
LIN {X 0,Y 134.686,Z 431.071,A -85,B 0,C 180,E1 -25376.26,E2 -25376.26} C_VEL
LIN {X 0,Y 134.405,Z 430.793,A -85,B 0,C 180,E1 -25380,E2 -25380} C_VEL
LIN {X 0,Y 134.703,Z 431.185,A -85,B 0,C 180,E1 -25384.301,E2 -25384.301} C_VEL
LIN {X 0,Y 137,Z 435.699,A -85,B 0,C 180,E1 -25392.593,E2 -25392.593} C_VEL
LIN {X 0,Y 138.813,Z 437.022,A -85,B 0,C 180,E1 -25395.881,E2 -25395.881} C_VEL
LIN {X 0,Y 140.835,Z 440.439,A -85,B 0,C 180,E1 -25399.116,E2 -25399.116} C_VEL
LIN {X 0,Y 142.755,Z 442.404,A -85,B 0,C 180,E1 -25401.516,E2 -25401.516} C_VEL
LIN {X 0,Y 145.368,Z 446.098,A -85,B 0,C 180,E1 -25404.454,E2 -25404.454} C_VEL
LIN {X 0,Y 146.59,Z 447.682,A -85,B 0,C 180,E1 -25405.67,E2 -25405.67} C_VEL
LIN {X 0,Y 149.941,Z 452.496,A -85,B 0,C 180,E1 -25408.714,E2 -25408.714} C_VEL
LIN {X 0,Y 154.159,Z 458.757,A -85,B 0,C 180,E1 -25412.023,E2 -25412.023} C_VEL
LIN {X 0,Y 159.816,Z 468.413,A -85,B 0,C 180,E1 -25415.888,E2 -25415.888} C_VEL
LIN {X 0,Y 164.555,Z 477.501,A -85,B 0,C 180,E1 -25418.752,E2 -25418.752} C_VEL
LIN {X 0,Y 166.081,Z 481.591,A -85,B 0,C 180,E1 -25419.68,E2 -25419.68} C_VEL
LIN {X 0,Y 163.601,Z 514.22,A -85,B 0,C 180,E1 -25420.871,E2 -25420.871} C_VEL
LIN {X 0,Y 161.865,Z 526.942,A -85,B 0,C 180,E1 -25421.616,E2 -25421.616} C_VEL
LIN {X 0,Y 159.408,Z 538.537,A -85,B 0,C 180,E1 -25422.632,E2 -25422.632} C_VEL
LIN {X 0,Y 156.366,Z 549.71,A -85,B 0,C 180,E1 -25424.017,E2 -25424.017} C_VEL
LIN {X 0,Y 152.015,Z 562.2,A -85,B 0,C 180,E1 -25426.094,E2 -25426.094} C_VEL
LIN {X 0,Y 147.388,Z 573.13,A -85,B 0,C 180,E1 -25428.578,E2 -25428.578} C_VEL
LIN {X 0,Y 143.008,Z 582.019,A -85,B 0,C 180,E1 -25431.202,E2 -25431.202} C_VEL
LIN {X 0,Y 138.235,Z 590.863,A -85,B 0,C 180,E1 -25434.639,E2 -25434.639} C_VEL
LIN {X 0,Y 133.828,Z 598.162,A -85,B 0,C 180,E1 -25438.322,E2 -25438.322} C_VEL
LIN {X 0,Y 129.55,Z 604.573,A -85,B 0,C 180,E1 -25442.541,E2 -25442.541} C_VEL
LIN {X 0,Y 125.999,Z 609.657,A -85,B 0,C 180,E1 -25447.018,E2 -25447.018} C_VEL
LIN {X 0,Y 123.218,Z 613.602,A -85,B 0,C 180,E1 -25451.718,E2 -25451.718} C_VEL
LIN {X 0,Y 121.249,Z 616.511,A -85,B 0,C 180,E1 -25456.594,E2 -25456.594} C_VEL
LIN {X 0,Y 119.695,Z 618.888,A -85,B 0,C 180,E1 -25463.257,E2 -25463.257} C_VEL
LIN {X 0,Y 119.432,Z 619.492,A -85,B 0,C 180,E1 -25466.627,E2 -25466.627} C_VEL
LIN {X 0,Y 119.363,Z 619.717,A -85,B 0,C 180,E1 -25470.001,E2 -25470.001} C_VEL
LIN {X 0,Y 119.432,Z 619.521,A -85,B 0,C 180,E1 -25473.374,E2 -25473.374} C_VEL
LIN {X 0,Y 120.282,Z 617.966,A -85,B 0,C 180,E1 -25480.096,E2 -25480.096} C_VEL
LIN {X 0,Y 121.248,Z 616.605,A -85,B 0,C 180,E1 -25483.407,E2 -25483.407} C_VEL
LIN {X 0,Y 123.198,Z 613.733,A -85,B 0,C 180,E1 -25488.286,E2 -25488.286} C_VEL
